(* CODESYS project CtaSysIO_2.0.0.0.library
   Description: Io System Library der CTA
   Version: 2.0.0.0
   Title: CtaSysIO
   Author: SIS
   DocFormat: reStructuredText
   LanguageModelAttribute: qualified-access-only
   Placeholder: CtaSysIO
   CompiledLibraryCompatibilityVersion: CODESYS V3.5 SP16 Patch 3
   Company: CTA
   DefaultNamespace: CtaSysIO

Project tree, tasks and I/O mapping:
  libraries: Standard, 3.5.18.0 (System); VisuDialogs, * (System); CtaSysConfig, 2.0.0.0 (CTA); CtaVisSymbols, 2.0.0.0 (CTA); VisuSymbols, 4.5.0.0 (System); CtaAppReport, 2.0.0.0 (CTA); CtaAppBmk, 2.0.0.0 (CTA); CtaVisHelp, 1.0.0.0 (CTA); CtaAppInfluxLog, 1.0.0.1 (CTA); SysCom, 3.5.17.0 (System); CtaAppBasic, 1.0.0.0 (CTA); Visu Utils, 4.5.0.0 (System)
  40 Visualizations/
    IO_FB/
      AI/
        visualisation SimAI_Temp
        visualisation SimAI
        visualisation SimAI_Temp_Querry
      AO/
        visualisation SimAO_Temp
        visualisation SimAO
        visualisation SimAO_Temp_Querry
      DI/
        visualisation SimDI
        visualisation SimDI_Temp
        visualisation SimDI_Temp_Querry
        SimValue/
          visualisation SimDI_Value
          visualisation SimDI_Value_Query
      DO/
        visualisation SimDO_Temp
        visualisation SimDO
        visualisation SimDO_Temp_Querry
        SimValue/
          visualisation SimDO_Value
          visualisation SimDO_Value_Query
      Simulation/
        visualisation Simulation
        visualisation ModulInfos
        visualisation SimulationInfos
        visualisation DIA_IO_CONFIG
      Parameter/
        visualisation VIS_IO_PARAMETER_BASE
        Parameter_AI/
          visualisation VIS_PARAMETER_AI
          visualisation VIS_PARAMETER_TEMP_AI
        Parameter_DI/
          visualisation VIS_PARAMETER_DI
          visualisation VIS_PARAMETER_TEMP_DI
        Parameter_AO/
          visualisation VIS_PARAMETER_AO
          visualisation VIS_PARAMETER_TEMP_AO
        Parameter_DO/
          visualisation VIS_PARAMETER_DO
          visualisation VIS_PARAMETER_TEMP_DO
      IO/
        visualisation SimIO
        visualisation SimIO_Query
        Invert/
          visualisation SimInvert
          visualisation SimInvert_Query
        visualisation SimIO_Temp
    IO_MANAGER/
      DEVICE/
        visualisation VIS_DEVICE
        visualisation VIS_DEVICE_QUERY
      visualisation DIA_IO_DEVICES
      NETZWERK/
        visualisation VIS_IO_DEVICES
        visualisation VIS_IO_DEVICES_NETWORK
    IO_TABLE/
      visualisation VIS_IO_TABLE
      visualisation VIS_IO_TABLE_QUERY
    IO_SLOT/
      visualisation VIS_IO_SLOT_IOS_ARRAY
      visualisation VIS_IO_SLOT_IOS_QUERY
      visualisation VIS_IO_SLOT_IOS
  30 Program Organization Units/
    IO_FB/
      IO/
        function block FB_IO [ST]: SELF, P_scfbIO_fbxSimulationLock, P_scfbIO_Simulation, ProSetInstancePathOnDynCreate, SELFPOINTER, IO_TYPE, IO_NR, PARENT, proSimVisu, proOK, proOkVisu, proPhysikalValueVisu, proIsSimLocked, proIsBOOL_IO, ADD_HAND, proLogName, DESTROY, BIG_SYBIL, LOW_SYBIL, SLOT_NR, REM_HAND
        function block FB_IO_TABLE [ST]: IO_NR, IO_TYPE, proSimVisu, SLOT_NR, proOkVisu, proPhysikalValueVisu
      AI/
        function block FB_AI [ST]: P_scfbAI_fbstPhysicalUnit, P_scfbAI_fbrMax, P_scfbAI_fbrMinPhysical, P_scfbAI_fbrMin, P_scfbAI_fbrPhysicalAlarm, P_scfbAI_fbrSimulationValue, P_scfbAI_fbrCorrectionValue, P_All_Init, proIsBOOL_IO, proPhysikalValueVisu, proPhysicalValue, proValue, metCyclicIoUpdate, metTrendLog, proAlUeberlauf, metConfig, proAlUnterlauf
      DO/
        function block FB_DO [ST]: P_scfbDO_fbxInvert, P_All_Init, P_scfbDO_fbxSimulationValue, metConfig, metTrendLog, proPhysikalValueVisu, proIsBOOL_IO, proValue, metCyclicIoUpdate
      AO/
        function block FB_AO [ST]: proIsBOOL_IO, P_All_Init, P_scfbAO_fbrMin, P_scfbAO_fbrMax, P_scfbAO_fbrSimulationValue, P_scfbAO_fbrMinPhysical, proValue, metCyclicIoUpdate, metTrendLog, metConfig, proPhysicalValue, proPhysikalValueVisu
      DI/
        function block FB_DI [ST]: metConfig, proPhysikalValueVisu, metCyclicIoUpdate, metTrendLog, P_scfbDI_fbxSimulationValue, P_scfbDI_fbxInvert, P_All_Init, proValue, proIsBOOL_IO
      FC/
        function fcScaleOut [ST]
        function fcScaleIn [ST]
    IO_DEVICE/
      function block FB_IO_DEVICE [ST]: AY_ITF_SLOT_VIS, BIG_SYBIL, LOW_SYBIL, ADDITION_DYN_SIZE, proVISU_DIA_NAME, IMAGE, COUNT, SELF, ADD_ERROR, ADD_SLOT, RELOAD_ARRAY, CHECK_IF_SLOT_EXIST, DEV_NR, DYN_SIZE, INSTANCE_PATH, ERROR, CREATE_SLOT, GET_SLOT, GET_IO, CHECK_ERROR, CHECK_HAND, ADD_HAND, HAND, REM_ERROR, REM_HAND, GET_STATE_READY_TO_SET_CONFIG, SET_STATE_READY_TO_SET_CONFIG, CHECK_SLOT, CONFIG_DONE, CHECK_SLOT_FAILS, SIM_IO_UPDATE, SIMULATION_ENABLED, FB_INIT, SIM_IO_TYPE
    IO_SLOT/
      function block FB_IO_SLOT [ST]: ADD_IO, CHECK_IF_IO_EXIST, CREATE_IO, GET_IO, BIG_SYBIL, LOW_SYBIL, PARENT, SELF, SLOT_NR, IMAGE, DYN_SIZE, RELOAD_ARRAY, AY_ITF_IO_VIS, SELFPOINTER, COUNT, ADD_ERROR, CHECK_SLOT
    IO_MANAGER/
      function block FB_IO_MANAGER [ST]: GET_DEVICE, GET_IO, AY_ITF_DEVICE_VIS, COUNT, ADD_DEVICE, CHECK_IF_DEVICE_EXIST, IMAGE, CHECK_SLOT
    FC/
      function FC_VIS_IO_TABLE [ST]
  00000000-0000-0000-0000-000000000000|D:\CoDeSys\LibrariesV3\trunk\Intern\CAA\CAA Template\3.4.0.0 draft\Placeholder.xml
  00000000-0000-0000-0000-000000000000|D:\CoDeSys\LibrariesV3\trunk\Intern\CAA\CAA Template\3.2.0.3 draft\Prefix.pdf
  00000000-0000-0000-0000-000000000000|D:\CoDeSys\LibrariesV3\trunk\Intern\CAA\CAA Template\3.5.2.0 draft\Placeholder.xml
  20 Structs/
    Parameter/
      data type scDI_Para
      data type scDO_Para
      data type scAI_Para
      data type scAO_Para
    data type enIOType
    data type enCheckIo
  50 Images/
  10 Documenation/
    global variables VersionHistory
    global variables readMe
  21 Interface/
    IO_MANAGER/
      interface ITF_IO_MANAGER: IMAGE, AY_ITF_DEVICE_VIS, COUNT
    IO_SLOT/
      interface ITF_IO_SLOT: BIG_SYBIL, LOW_SYBIL, SELF, PARENT, SLOT_NR, IMAGE, DYN_SIZE, GET_IO, CREATE_IO, AY_ITF_IO_VIS, RELOAD_ARRAY, SELFPOINTER, COUNT, CHECK_SLOT
    IO_DEVICE/
      interface ITF_IO_DEVICE: INSTANCE_PATH, ADD_ERROR, LOW_SYBIL, ERROR, ADD_HAND, SELF, HAND, IMAGE, DEV_NR, DYN_SIZE, RELOAD_ARRAY, COUNT, GET_IO, BIG_SYBIL, ADDITION_DYN_SIZE, proVISU_DIA_NAME, AY_ITF_SLOT_VIS, REM_ERROR, REM_HAND, GET_STATE_READY_TO_SET_CONFIG, SET_STATE_READY_TO_SET_CONFIG, CHECK_SLOT, SIM_IO_TYPE
    IO_FB/
      AI/
        interface ITF_AI: P_scfbAI_fbrPhysicalAlarm, P_scfbAI_fbrSimulationValue, P_scfbAI_fbstPhysicalUnit, P_scfbAI_fbrCorrectionValue, P_scfbAI_fbrMax, P_scfbAI_fbrMin, P_scfbAI_fbrMinPhysical, P_All_Init, proAlUeberlauf, proValue, proAlUnterlauf, metCyclicIoUpdate, proPhysicalValue
      AO/
        interface ITF_AO: proValue, proPhysicalValue, P_scfbAO_fbrMax, P_scfbAO_fbrMin, P_scfbAO_fbrMinPhysical, P_scfbAO_fbrSimulationValue, P_All_Init, metCyclicIoUpdate
      DI/
        interface ITF_DI: metCyclicIoUpdate, P_scfbDI_fbxInvert, P_scfbDI_fbxSimulationValue, P_All_Init, proValue
      DO/
        interface ITF_DO: proValue, metCyclicIoUpdate, P_scfbDO_fbxSimulationValue, P_All_Init, P_scfbDO_fbxInvert
      IO/
        interface ITF_IO: proIsBOOL_IO, P_scfbIO_Simulation, P_scfbIO_fbxSimulationLock, BIG_SYBIL, SELF, PARENT, IO_TYPE, proOK, ProSetInstancePathOnDynCreate, LOW_SYBIL, proOkVisu, IO_NR, SELFPOINTER, proPhysikalValueVisu, proSimVisu, proIsSimLocked, proLogName
        interface ITF_IO_TABLE: IO_TYPE, IO_NR, SLOT_NR, proOkVisu, proPhysikalValueVisu, proSimVisu
  11 Library Parameter/
    global variables Parameter
  12 Konstanten/
    global variables GlobalKonstant
  60 Textlisten/
    text list txtIOType
    text list txtWarning
    text list txtError
    text list txtPhysicalUnit
  13 Globale Variablen/
    global variables GVL_IO
  text list GlobalTextList
  5ce3da45-db07-42e7-a21c-a00fff4ed8f6|S:\_Temporär_SIS\CtaCodesysLibrary\01_Library\CtaSysIO\04_Image\0750_432.bmp
  5ce3da45-db07-42e7-a21c-a00fff4ed8f6|S:\_Temporär_SIS\CtaCodesysLibrary\01_Library\CtaSysIO\04_Image\0750_455.bmp
  5ce3da45-db07-42e7-a21c-a00fff4ed8f6|S:\_Temporär_SIS\CtaCodesysLibrary\01_Library\CtaSysIO\04_Image\0750_466.bmp
  5ce3da45-db07-42e7-a21c-a00fff4ed8f6|S:\_Temporär_SIS\CtaCodesysLibrary\01_Library\CtaSysIO\04_Image\0750_597.bmp
  5ce3da45-db07-42e7-a21c-a00fff4ed8f6|S:\_Temporär_SIS\CtaCodesysLibrary\01_Library\CtaSysIO\04_Image\0750_652.bmp
  5ce3da45-db07-42e7-a21c-a00fff4ed8f6|S:\_Temporär_SIS\CtaCodesysLibrary\01_Library\CtaSysIO\04_Image\0750_1415.bmp
  5ce3da45-db07-42e7-a21c-a00fff4ed8f6|S:\_Temporär_SIS\CtaCodesysLibrary\01_Library\CtaSysIO\04_Image\0750_8212.bmp
  5ce3da45-db07-42e7-a21c-a00fff4ed8f6|S:\_Temporär_SIS\CtaCodesysLibrary\01_Library\CtaSysIO\04_Image\0750_555.bmp
*)

// 20 Structs/Parameter/scDI_Para
TYPE scDI_Para :
	STRUCT
		xSimulationLock		:	BOOL;
		xInvert				:	BOOL;
	END_STRUCT
END_TYPE

// 20 Structs/Parameter/scDO_Para
TYPE scDO_Para :
	STRUCT
		xSimulationLock		:	BOOL;
		xInvert				:	BOOL;
	END_STRUCT
END_TYPE

// 20 Structs/Parameter/scAI_Para
TYPE scAI_Para :
	STRUCT
		xSimulationLock		:	BOOL;
		rMin				:	REAL;
		rMax				:	REAL;
		rMinPhysical		:	REAL;
		rPhysicalAlarm		:	REAL;
		rCorrectionValue	:	REAL;
		stPhysicalUnit		:	STRING(40);
	END_STRUCT
END_TYPE

// 20 Structs/Parameter/scAO_Para
TYPE scAO_Para :
	STRUCT
		xSimulationLock		:	BOOL;
		rMin				:	REAL;
		rMax				:	REAL;
		rMinPhysical		:	REAL;
	END_STRUCT
END_TYPE

// 20 Structs/enIOType
{attribute 'qualified_only'}
{attribute 'to_string'}

TYPE enIOType :
(
	Unknown 		:= 0,
	Digital_IN		:= 1,
	Digital_OUT		:= 2,	
	DC_0_10V_OUT	:= 3,
	DC_4_20mA_OUT	:= 4,
	DC_0_10V_IN		:= 5,
	DC_4_20mA_IN	:= 6,
	OHM				:= 7,
	DC_0_20mA_OUT	:= 8,
	TEMPERATUR		:= 9,
	DC_0_20mA_IN	:= 10
);
END_TYPE

// 20 Structs/enCheckIo
TYPE enCheckIo :
(
		DI_IO	:=	0,
		AI_IO	:=	1,
		DO_IO	:=	2,
		AO_IO	:=	3
);
END_TYPE

// 10 Documenation/VersionHistory
(* 

.. image:: ../../Images/CTA_Logo.jpg
   :align: right
   :width: 15% 

**Vorlage**   


============ =========== =========== ============================================
**Date**     **Version** **Author**  **Change**
------------ ----------- ----------- --------------------------------------------
04.03.2021   0.0.0.0     SIS         Vorlage erstellt

============ =========== =========== ============================================


*)
VAR_GLOBAL
    stInfo : STRING:= '0.0.0.0, Vorlage, CTA';
END_VAR

// 10 Documenation/readMe
(*

**ReadMe**
 
|	**Empfehlung**
|
|	Dokumentrieren Sie die Library für eine nachhaltige Entwicklung
|     
| *Beispiel*
| 
| Dies ist die Vorlage Library der CTA. Erstellen Sie ihre Library anhand dieser Vorlage.
*)

VAR_GLOBAL
    xReadMeDone              :   BOOL;
END_VAR

// 13 Globale Variablen/GVL_IO
{attribute 'qualified_only'}
VAR_GLOBAL	
	FB_IO_MANAGER : FB_IO_MANAGER;
END_VAR

// 11 Library Parameter/Parameter
{attribute 'qualified_only'}
VAR_GLOBAL CONSTANT
	SPS_BMK_ID        		: STRING(20)   := 'SPS';
	MAX_NUM_OF_DI			: INT := 200;
	MAX_NUM_OF_DO			: INT := 200;
	MAX_NUM_OF_AI			: INT := 100;
	MAX_NUM_OF_AO			: INT := 100;	
	                		
	MAX_NUM_OF_IOS			: INT := MAX_NUM_OF_DI + MAX_NUM_OF_DO + MAX_NUM_OF_AI + MAX_NUM_OF_AO;
	
	MAX_NUM_OF_COMTYPES		: INT := 10;
END_VAR

// 12 Konstanten/GlobalKonstant
{attribute 'qualified_only'}
VAR_GLOBAL CONSTANT
    stWarningTextList   :   STRING  := 'CtaSysIO.txtWarning';
    stErrorTextList     :   STRING  := 'CtaSysIO.txtError';
END_VAR

// 30 Program Organization Units/IO_DEVICE/FB_IO_DEVICE
{attribute 'reflection'}
FUNCTION_BLOCK FB_IO_DEVICE EXTENDS CtaAppBmk.fbBMK IMPLEMENTS ITF_IO_DEVICE
VAR_INPUT
	usiDevNr	:	USINT;
END_VAR
VAR_OUTPUT
	xReadyToIoConfig			:	BOOL;
	xConfigDone					:	BOOL;
	xError						:	BOOL;
	xSlotMissmatch				:	BOOL;
	xHand						:	BOOL;
	udiDynMem					:	UDINT;	
END_VAR
VAR
	_IMAGE						:	STRING;
	
	_ITF_BIG_SYBIL				:	ITF_IO_DEVICE;
	_ITF_LOW_SYBIL				:	ITF_IO_DEVICE;
	                			
	_BASE_SLOT					:	ITF_IO_SLOT;
	_TEMP_REG_SLOT				:	ITF_IO_SLOT;
	_NEXT_SLOT_LAST_GET			:	ITF_IO_SLOT;	
	
	_COUNT						:	UINT;
	_udiDynMemTemp				:	UDINT;	
	_ayITF_SLOTS				:	ARRAY[0..255] OF ITF_IO_SLOT;
	_ayITF_SLOT_VIS				:	ARRAY[1..10] OF ITF_IO_SLOT;
	
	_ALLOW_SIMULATION			:	BOOL;
	_ENABLE_SIMULATION			:	BOOL;
	_INIT_DONE_SIMULATION		:	BOOL;
	
	udiCountError				:	UDINT;	
	udiCountHand				:	UDINT;
	udiCountCheckSlotFails		:	UDINT;
	udiCountCheckSlotFailsOld	:	UDINT;
	
END_VAR

xSlotMissmatch 	:= CHECK_SLOT_FAILS();
xHand 			:= CHECK_HAND();
xError 			:= CHECK_ERROR();

SIM_IO_UPDATE();

PROPERTY AY_ITF_SLOT_VIS : ARRAY[1..10] OF ITF_IO_SLOT;
GET
AY_ITF_SLOT_VIS := _ayITF_SLOT_VIS;
END_GET
END_PROPERTY

{attribute 'estimated-stack-usage' := '104'}
PROPERTY BIG_SYBIL : ITF_IO_DEVICE
SET
_ITF_BIG_SYBIL := BIG_SYBIL;
IF __QUERYINTERFACE(_ITF_BIG_SYBIL,_ITF_BIG_SYBIL) THEN
	IF _ITF_BIG_SYBIL.LOW_SYBIL <> SELF THEN
		_ITF_BIG_SYBIL.LOW_SYBIL := THIS^;
	END_IF;
END_IF;
END_SET
GET
BIG_SYBIL := _ITF_BIG_SYBIL;
END_GET
END_PROPERTY

{attribute 'estimated-stack-usage' := '104'}
PROPERTY LOW_SYBIL : ITF_IO_DEVICE
GET
LOW_SYBIL := _ITF_LOW_SYBIL;
END_GET
SET
_ITF_LOW_SYBIL := LOW_SYBIL;
IF __QUERYINTERFACE(_ITF_LOW_SYBIL,_ITF_LOW_SYBIL) THEN
	IF _ITF_LOW_SYBIL.BIG_SYBIL <> SELF THEN
		_ITF_LOW_SYBIL.BIG_SYBIL := THIS^;
	END_IF;
END_IF;
END_SET
END_PROPERTY

PROPERTY ADDITION_DYN_SIZE : DINT
SET
VAR
	diTemp	:	DINT;
END_VAR
IF ADDITION_DYN_SIZE > 0 THEN
	_udiDynMemTemp := _udiDynMemTemp + TO_UDINT(ADDITION_DYN_SIZE);
ELSE
	_udiDynMemTemp := _udiDynMemTemp - TO_UDINT(ADDITION_DYN_SIZE);
END_IF;
udiDynMem	:= MAX(udiDynMem,_udiDynMemTemp);
END_SET
END_PROPERTY

PROPERTY proVISU_DIA_NAME : STRING
GET
proVISU_DIA_NAME := '';
END_GET
END_PROPERTY

PROPERTY IMAGE : STRING
GET
IMAGE := _IMAGE;
END_GET
SET
_IMAGE := IMAGE;
END_SET
END_PROPERTY

PROPERTY COUNT : UINT
GET
COUNT := _COUNT;
END_GET
END_PROPERTY

PROPERTY SELF : ITF_IO_DEVICE
GET
SELF := THIS^;
END_GET
END_PROPERTY

METHOD ADD_ERROR
VAR_INPUT
END_VAR
udiCountError := udiCountError + 1;
END_METHOD

METHOD ADD_SLOT
VAR_INPUT
	ITF_SLOT_IN		:	ITF_IO_SLOT;
END_VAR
VAR
	ITF_TEMP		:	ITF_IO_SLOT;
	ITF_TEMP_BIG	:	ITF_IO_SLOT;
	ITF_TEMP_LOW	:	ITF_IO_SLOT;
	xDone			:	BOOL;
END_VAR
(* Check if Valid Interface Input *)
IF __QUERYINTERFACE(ITF_SLOT_IN,ITF_SLOT_IN) THEN
	ITF_SLOT_IN.PARENT := THIS^;
	IF TO_DINT(ITF_SLOT_IN.SLOT_NR) >= LOWER_BOUND(_ayITF_SLOTS,1) AND
	   TO_DINT(ITF_SLOT_IN.SLOT_NR) <= UPPER_BOUND(_ayITF_SLOTS,1) THEN
	   _ayITF_SLOTS[ITF_SLOT_IN.SLOT_NR] := ITF_SLOT_IN;
	END_IF;
	(* Check if Valid Interface Base*)
	IF __QUERYINTERFACE(_BASE_SLOT,_BASE_SLOT) THEN
		(* Check if Valid Interface Temporary registration *)
		IF __QUERYINTERFACE(_TEMP_REG_SLOT,ITF_TEMP) THEN
			REPEAT
				(* Get Big Sybil of registration *)
				IF __QUERYINTERFACE(ITF_TEMP.BIG_SYBIL,ITF_TEMP_BIG) THEN
					(* Check if Adress is Lower *)
					IF ITF_SLOT_IN.SLOT_NR <= ITF_TEMP.SLOT_NR THEN
						(* Check if Adress is Bigger and update if yes*)
						IF ITF_SLOT_IN.SLOT_NR >= ITF_TEMP_BIG.SLOT_NR THEN
							ITF_SLOT_IN.BIG_SYBIL := ITF_TEMP.BIG_SYBIL;
							ITF_SLOT_IN.LOW_SYBIL := ITF_TEMP;
							xDone	 := TRUE;							
						END_IF;
					(* Adress is Bigger update *)
					ELSE
						IF __QUERYINTERFACE(ITF_TEMP.LOW_SYBIL,ITF_TEMP_LOW) THEN
							IF 	ITF_SLOT_IN.SLOT_NR <= ITF_TEMP_LOW.SLOT_NR THEN
								ITF_SLOT_IN.LOW_SYBIL := ITF_TEMP.LOW_SYBIL;
								ITF_SLOT_IN.BIG_SYBIL := ITF_TEMP;
								xDone	 := TRUE;
							END_IF;
						ELSE
							ITF_SLOT_IN.LOW_SYBIL := ITF_TEMP.LOW_SYBIL;
							ITF_SLOT_IN.BIG_SYBIL := ITF_TEMP;
							xDone	 := TRUE;
							(* Update Registation Job if temp is the last one *)
							IF ITF_TEMP = _TEMP_REG_SLOT THEN
								_TEMP_REG_SLOT := ITF_SLOT_IN;
								_TEMP_REG_SLOT.LOW_SYBIL := 0;
							END_IF;
						END_IF;
					END_IF;
				(* Interface is same as the Base*)
				ELSIF ITF_TEMP = _BASE_SLOT THEN
					(* Check if the Input Interface needs to be the new base*)
					IF ITF_SLOT_IN.SLOT_NR <= ITF_TEMP.SLOT_NR THEN 
						ITF_SLOT_IN.LOW_SYBIL := ITF_TEMP;
						_BASE_SLOT 				:= ITF_SLOT_IN;
						_BASE_SLOT.BIG_SYBIL 	:= 0;
						xDone	 				:= TRUE; 
					ELSE
						(* Update Registation Job if temp is the last one *)
						IF ITF_TEMP = _TEMP_REG_SLOT THEN
							_TEMP_REG_SLOT				:= ITF_SLOT_IN;
							_TEMP_REG_SLOT.LOW_SYBIL 	:= 0;
						END_IF
						ITF_SLOT_IN.LOW_SYBIL := _BASE_SLOT.LOW_SYBIL;
						_BASE_SLOT.LOW_SYBIL 	:= ITF_SLOT_IN;
					END_IF;
				END_IF;
				(* Get Next Interface to Check*)
				__QUERYINTERFACE(ITF_TEMP.BIG_SYBIL,ITF_TEMP);
			UNTIL xDone OR ITF_TEMP = 0 
			END_REPEAT
		ELSE
			(* Set Base Low sybill on second call*)
			_BASE_SLOT.LOW_SYBIL 	:= ITF_SLOT_IN;
			_TEMP_REG_SLOT			:= ITF_SLOT_IN;		
		END_IF;		
	ELSE
		(* Set Base on first call*)
		_BASE_SLOT 		:= ITF_SLOT_IN;
		_TEMP_REG_SLOT 	:= ITF_SLOT_IN;
	END_IF;
	(* Count Jobs *)
	_COUNT := _COUNT + 1;
	THIS^.RELOAD_ARRAY(TRUE,FALSE,FALSE);
END_IF;
END_METHOD

METHOD RELOAD_ARRAY
VAR_INPUT
	xInit	: BOOL;
	xLoadNext10	: BOOL;
	xLoadLast10	: BOOL;
END_VAR
VAR
	diFor				:	DINT;
	ITF_TEMP_CLIENT_VIS	:	ITF_IO_SLOT;
	ITF_TEMP_SAFE		:	ITF_IO_SLOT;
	ITF_TEMP_LAST_VALID	:	ITF_IO_SLOT;
END_VAR
(* Init Array *)
IF xInit THEN
	_ayITF_SLOT_VIS[LOWER_BOUND(_ayITF_SLOT_VIS,1)] := _BASE_SLOT;
	FOR diFor := LOWER_BOUND(_ayITF_SLOT_VIS,1) TO UPPER_BOUND(_ayITF_SLOT_VIS,1) -1 DO
		IF __QUERYINTERFACE(_ayITF_SLOT_VIS[diFor],ITF_TEMP_CLIENT_VIS) THEN
			_ayITF_SLOT_VIS[diFor + 1]	:= _ayITF_SLOT_VIS[diFor].LOW_SYBIL;
		ELSE
			_ayITF_SLOT_VIS[diFor + 1] := 0;
		END_IF;	
	END_FOR;
(* Load Next 10 *)
ELSIF xLoadNext10 THEN
	IF __QUERYINTERFACE(_ayITF_SLOT_VIS[UPPER_BOUND(_ayITF_SLOT_VIS,1)],ITF_TEMP_CLIENT_VIS) THEN
		_ayITF_SLOT_VIS[LOWER_BOUND(_ayITF_SLOT_VIS,1)] := ITF_TEMP_CLIENT_VIS.LOW_SYBIL;
		FOR diFor := LOWER_BOUND(_ayITF_SLOT_VIS,1) TO UPPER_BOUND(_ayITF_SLOT_VIS,1) -1 DO
			IF __QUERYINTERFACE(_ayITF_SLOT_VIS[diFor],ITF_TEMP_CLIENT_VIS) THEN
				_ayITF_SLOT_VIS[diFor + 1]	:= _ayITF_SLOT_VIS[diFor].LOW_SYBIL;
			ELSE
				_ayITF_SLOT_VIS[diFor + 1] := 0;
			END_IF;	
		END_FOR;
	END_IF;
(* Load Last 10 *)
ELSIF xLoadLast10 THEN
	IF __QUERYINTERFACE(_ayITF_SLOT_VIS[LOWER_BOUND(_ayITF_SLOT_VIS,1)],ITF_TEMP_CLIENT_VIS) THEN
		IF __QUERYINTERFACE(_ayITF_SLOT_VIS[LOWER_BOUND(_ayITF_SLOT_VIS,1)].BIG_SYBIL,ITF_TEMP_SAFE) THEN
			_ayITF_SLOT_VIS[UPPER_BOUND(_ayITF_SLOT_VIS,1)] := ITF_TEMP_CLIENT_VIS.BIG_SYBIL;
			FOR diFor := UPPER_BOUND(_ayITF_SLOT_VIS,1) TO LOWER_BOUND(_ayITF_SLOT_VIS,1) + 1 BY -1 DO 
				IF __QUERYINTERFACE(_ayITF_SLOT_VIS[diFor],ITF_TEMP_CLIENT_VIS) THEN
					ITF_TEMP_LAST_VALID  			:= _ayITF_SLOT_VIS[diFor];
					_ayITF_SLOT_VIS[diFor - 1]	:= _ayITF_SLOT_VIS[diFor].BIG_SYBIL;
				ELSE
					(* Resort if new ones Inside *)
					_ayITF_SLOT_VIS[LOWER_BOUND(_ayITF_SLOT_VIS,1)] := ITF_TEMP_LAST_VALID;
					FOR diFor := LOWER_BOUND(_ayITF_SLOT_VIS,1) TO UPPER_BOUND(_ayITF_SLOT_VIS,1) -1 DO
						IF __QUERYINTERFACE(_ayITF_SLOT_VIS[diFor],ITF_TEMP_CLIENT_VIS) THEN
							_ayITF_SLOT_VIS[diFor + 1]	:= _ayITF_SLOT_VIS[diFor].LOW_SYBIL;
						ELSE
							_ayITF_SLOT_VIS[diFor + 1] := 0;
						END_IF;	
					END_FOR;					
				END_IF;	
			END_FOR;
		END_IF;
	END_IF;	
END_IF;
END_METHOD

METHOD CHECK_IF_SLOT_EXIST : BOOL
VAR_INPUT
	_usiSlotNr			: 	USINT;
END_VAR
VAR
	_TEMP_CHK_SLOT	:	ITF_IO_SLOT;
	udiSafe			:	UDINT;
END_VAR
IF __QUERYINTERFACE(_BASE_SLOT,_TEMP_CHK_SLOT) THEN
	REPEAT 
		IF _TEMP_CHK_SLOT.SLOT_NR = _usiSlotNr THEN
			CHECK_IF_SLOT_EXIST := TRUE;
		END_IF;
		_TEMP_CHK_SLOT := _TEMP_CHK_SLOT.LOW_SYBIL;
		udiSafe	:= udiSafe + 1;
	UNTIL CHECK_IF_SLOT_EXIST OR _TEMP_CHK_SLOT = 0 OR udiSafe >= 16#FFFFFFFE
	END_REPEAT
ELSE
	CHECK_IF_SLOT_EXIST := FALSE;
END_IF
END_METHOD

PROPERTY DEV_NR : USINT
GET
DEV_NR := usiDevNr;
END_GET
END_PROPERTY

PROPERTY DYN_SIZE : UDINT
GET
DYN_SIZE := udiDynMem;
END_GET
END_PROPERTY

PROPERTY INSTANCE_PATH : STRING(255)
GET
INSTANCE_PATH := stInstancePath;
END_GET
END_PROPERTY

PROPERTY ERROR : BOOL
GET
ERROR := xError;
END_GET
END_PROPERTY

METHOD CREATE_SLOT : BOOL
VAR_INPUT
	_usiSlotNr			: 	USINT;
	_stSlotImage		:	STRING;
END_VAR
VAR	
	pFbIO				:	POINTER TO FB_IO_SLOT;
END_VAR
IF NOT CHECK_IF_SLOT_EXIST(_usiSlotNr) THEN
	pFbIO := __NEW(FB_IO_SLOT);
	IF pFbIO <> 0 THEN
		_udiDynMemTemp 							:= _udiDynMemTemp + SIZEOF(FB_IO);
		udiDynMem								:= MAX(udiDynMem,_udiDynMemTemp);
		pFbIO^.SLOT_NR		 					:= _usiSlotNr;
		pFbIO^.IMAGE		 					:= _stSlotImage;
		ADD_SLOT(pFbIO^);
	ELSE
		ADD_ERROR();
	END_IF;
END_IF;
END_METHOD

METHOD GET_SLOT : ITF_IO_SLOT
VAR_INPUT
	_usiSlotNr			: 	USINT;
END_VAR
VAR
	_TEMP_GET_SLOT	:	ITF_IO_SLOT;
	udiSafe			:	UDINT;
	xNextIoInUse	:	BOOL;
END_VAR
IF TO_DINT(_usiSlotNr) >= LOWER_BOUND(_ayITF_SLOTS,1) AND
   TO_DINT(_usiSlotNr) <= UPPER_BOUND(_ayITF_SLOTS,1) THEN
   GET_SLOT := _ayITF_SLOTS[_usiSlotNr];
END_IF;

IF GET_SLOT = 0 THEN
	IF __QUERYINTERFACE(_NEXT_SLOT_LAST_GET,_TEMP_GET_SLOT) THEN
		xNextIoInUse := TRUE;
	ELSIF __QUERYINTERFACE(_BASE_SLOT,_TEMP_GET_SLOT) THEN
		xNextIoInUse := FALSE;
	END_IF;
	
	IF __QUERYINTERFACE(_TEMP_GET_SLOT,_TEMP_GET_SLOT) THEN
		REPEAT 
			IF _TEMP_GET_SLOT.SLOT_NR = _usiSlotNr THEN
				GET_SLOT := _TEMP_GET_SLOT;
			END_IF;
			_TEMP_GET_SLOT	 	:= _TEMP_GET_SLOT.LOW_SYBIL;
			_NEXT_SLOT_LAST_GET	:= _TEMP_GET_SLOT;
			IF _TEMP_GET_SLOT = 0 AND xNextIoInUse THEN
				__QUERYINTERFACE(_BASE_SLOT,_TEMP_GET_SLOT);
				xNextIoInUse := FALSE;
			END_IF;
			udiSafe	:= udiSafe + 1;
		UNTIL GET_SLOT <> 0 OR _TEMP_GET_SLOT = 0 OR udiSafe >= 16#FFFFFFFE
		END_REPEAT
	ELSE
		GET_SLOT := 0;
	END_IF;
END_IF;
END_METHOD

METHOD GET_IO : ITF_IO
VAR_INPUT
	_usiSlotNr			: 	USINT;
	_usiIoNr			: 	USINT;
END_VAR	
VAR
	_TEMP_GET_SLOT	:	ITF_IO_SLOT;
	_TEMP_GET_IO		:	ITF_IO;
	udiSafe				:	UDINT;
END_VAR
IF __QUERYINTERFACE(GET_SLOT(_usiSlotNr),_TEMP_GET_SLOT) THEN
	GET_IO := _TEMP_GET_SLOT.GET_IO(_usiIoNr);
END_IF;
END_METHOD

METHOD CHECK_ERROR : BOOL
VAR_INPUT
END_VAR
CHECK_ERROR := udiCountError <> 0;
END_METHOD

METHOD CHECK_HAND : BOOL
VAR_INPUT
END_VAR
CHECK_HAND := udiCountHand <> 0;
END_METHOD

METHOD ADD_HAND
VAR_INPUT
END_VAR
udiCountHand := udiCountHand + 1;
END_METHOD

PROPERTY HAND : BOOL
GET
HAND := xHand;
END_GET
END_PROPERTY

METHOD REM_ERROR
VAR_INPUT
END_VAR
VAR
	ITF_IO_DEVICE_TEMP	:	ITF_IO_DEVICE;
END_VAR
udiCountError := udiCountError - 1;
END_METHOD

METHOD REM_HAND
VAR_INPUT
END_VAR
VAR
	ITF_IO_DEVICE_TEMP	:	ITF_IO_DEVICE;
END_VAR
udiCountHand := udiCountHand - 1;
END_METHOD

PROPERTY GET_STATE_READY_TO_SET_CONFIG : BOOL
GET
GET_STATE_READY_TO_SET_CONFIG := xReadyToIoConfig;
END_GET
END_PROPERTY

PROPERTY SET_STATE_READY_TO_SET_CONFIG : BOOL
SET
xReadyToIoConfig := SET_STATE_READY_TO_SET_CONFIG;
END_SET
END_PROPERTY

METHOD CHECK_SLOT : BOOL
VAR_INPUT
	_usiSlotNr		: 	USINT;
	enCheckIoIn		:	enCheckIo;
	usiAnzIoType	:	USINT;
END_VAR
VAR
	ITF_SLOT		: 	ITF_IO_SLOT;
END_VAR
ITF_SLOT := GET_SLOT(_usiSlotNr);
IF __QUERYINTERFACE(ITF_SLOT,ITF_SLOT) THEN
	CHECK_SLOT := ITF_SLOT.CHECK_SLOT(enCheckIoIn,usiAnzIoType);
ELSE
	CHECK_SLOT := FALSE;
END_IF;
IF NOT CHECK_SLOT AND xConfigDone THEN
	udiCountCheckSlotFails := udiCountCheckSlotFails + 1;
END_IF;
END_METHOD

PROPERTY CONFIG_DONE : BOOL
SET
xConfigDone := CONFIG_DONE;
END_SET
GET
CONFIG_DONE := xConfigDone;
END_GET
END_PROPERTY

METHOD INTERNAL CHECK_SLOT_FAILS : BOOL
VAR_INPUT
END_VAR
IF udiCountCheckSlotFails > 0 AND udiCountCheckSlotFails <> udiCountCheckSlotFailsOld THEN
	ADD_ERROR();
	udiCountCheckSlotFailsOld := udiCountCheckSlotFails;
ELSIF udiCountCheckSlotFails = 0 AND udiCountCheckSlotFails <> udiCountCheckSlotFailsOld THEN
	udiCountCheckSlotFailsOld := udiCountCheckSlotFails;
	REM_ERROR();
END_IF;
CHECK_SLOT_FAILS := udiCountCheckSlotFails > 0;
udiCountCheckSlotFails := 0;
END_METHOD

METHOD SIM_IO_UPDATE
VAR
	_ITF_SLOT_SIM	:	ITF_IO_SLOT;
	_ITF_IO_SIM		:	ITF_IO;
	_ITF_IO_SIM_DI	:	ITF_DI;
	_ITF_IO_SIM_AI	:	ITF_AI;
	_ITF_IO_SIM_DO	:	ITF_DO;
	_ITF_IO_SIM_AO	:	ITF_AO;
END_VAR
VAR
	usiFor			:	USINT;
END_VAR
// Prüfen, ob die Simulation aktiviert ist und die Initialisierung abgeschlossen wurde
IF SIMULATION_ENABLED AND CONFIG_DONE THEN

	// Prüfen, ob das Basismodul (_BASE_SLOT) das Interface für simulierte Slots (_ITF_SLOT_SIM) unterstützt
	IF __QUERYINTERFACE(_BASE_SLOT, _ITF_SLOT_SIM) THEN

		// Wiederhole, solange es noch simulierte Slots gibt
		REPEAT
			// Iteriere über alle IOs im aktuellen simulierten Slot
			FOR usiFor := 1 TO _ITF_SLOT_SIM.COUNT DO
				// Hole das IO-Element an der aktuellen Position
				_ITF_IO_SIM := _ITF_SLOT_SIM.GET_IO(usiFor);

				// Prüfen, ob es sich um ein digitales Eingangsmodul handelt
				IF __QUERYINTERFACE(_ITF_IO_SIM, _ITF_IO_SIM_DI) THEN
					// Zyklisches Update für digitales Eingangssignal ausführen
					_ITF_IO_SIM_DI.metCyclicIoUpdate(FALSE, TRUE);

				// Prüfen, ob es sich um ein analoges Eingangsmodul handelt
				ELSIF __QUERYINTERFACE(_ITF_IO_SIM, _ITF_IO_SIM_AI) THEN
					// Zyklisches Update für analoges Eingangssignal ausführen
					_ITF_IO_SIM_AI.metCyclicIoUpdate(TRUE, 0, FALSE, FALSE);

				// Prüfen, ob es sich um ein digitales Ausgangsmodul handelt
				ELSIF __QUERYINTERFACE(_ITF_IO_SIM, _ITF_IO_SIM_DO) THEN
					// Zyklisches Update für digitales Ausgangssignal ausführen
					_ITF_IO_SIM_DO.metCyclicIoUpdate(TRUE);

				// Prüfen, ob es sich um ein analoges Ausgangsmodul handelt
				ELSIF __QUERYINTERFACE(_ITF_IO_SIM, _ITF_IO_SIM_AO) THEN
					// Zyklisches Update für analoges Ausgangssignal ausführen
					_ITF_IO_SIM_AO.metCyclicIoUpdate(TRUE);
				END_IF;
			END_FOR;

			// Zum nächsten simulierten Slot wechseln (Linked-List-Mechanismus oder ähnliche Struktur)
			_ITF_SLOT_SIM := _ITF_SLOT_SIM.LOW_SYBIL;

		// Wiederhole solange, bis kein weiterer Slot vorhanden ist (d.h. Ende der Kette erreicht)
		UNTIL _ITF_SLOT_SIM = 0
		END_REPEAT;
	END_IF;
END_IF;;
END_METHOD

(* Enable Simulation *)
PROPERTY SIMULATION_ENABLED : BOOL
GET
SIMULATION_ENABLED := _ENABLE_SIMULATION;
END_GET
END_PROPERTY

//FB_Init ist immer implizit verfügbar und wird primär für die Initialisierung verwendet.
//Der Rückgabewert wird nicht ausgewertet. Für gezielte Einflussnahme können Sie
//die Methoden explizit deklarieren und darin mit dem Standard-Initialisierungscode 
//zusätzlichen Code bereitstellen. Sie können den Rückgabewert auswerten.
METHOD FB_Init: BOOL
VAR_INPUT    
	bInitRetains				: BOOL; // TRUE: Die Retain-Variablen werden initialisiert (Reset warm / Reset kalt)    
	bInCopyCode					: BOOL;  // TRUE: Die Instanz wird danach in den Kopiercode kopiert (Online-Change)
	xEnableSimulationOnReboot	: BOOL;
END_VAR
_ENABLE_SIMULATION := xEnableSimulationOnReboot;
END_METHOD

METHOD SIM_IO_TYPE
VAR_INPUT
	_usiSlotNr		: 	USINT;
	enSimIoTypeIn	:	enIOType;
	usiAnzIoType	:	USINT;
	_stSlotImage	:	STRING;
END_VAR
VAR
	usiFor			:	USINT;
	ITF_SLOT_TEMP	:	ITF_IO_SLOT;
END_VAR
IF SIMULATION_ENABLED THEN
	IF _usiSlotNr > _COUNT THEN
		CREATE_SLOT(_usiSlotNr,_stSlotImage);
		FOR usiFor := 1 TO usiAnzIoType DO
			ITF_SLOT_TEMP := GET_SLOT(_usiSlotNr);
			IF __QUERYINTERFACE(ITF_SLOT_TEMP,ITF_SLOT_TEMP) THEN
				ITF_SLOT_TEMP.CREATE_IO(usiFor,enSimIoTypeIn);
			END_IF;
		END_FOR;
	ELSE
		_INIT_DONE_SIMULATION := TRUE;
	END_IF;
END_IF;
END_METHOD

END_FUNCTION_BLOCK

// 21 Interface/IO_DEVICE/ITF_IO_DEVICE
INTERFACE ITF_IO_DEVICE EXTENDS CtaAppBmk.ITF_BMK

PROPERTY INSTANCE_PATH : STRING(255)
GET
END_GET
END_PROPERTY

METHOD ADD_ERROR
VAR_INPUT
END_VAR
END_METHOD

{attribute 'estimated-stack-usage' := '104'}
PROPERTY LOW_SYBIL : ITF_IO_DEVICE
SET
END_SET
GET
END_GET
END_PROPERTY

PROPERTY ERROR : BOOL
GET
END_GET
END_PROPERTY

METHOD ADD_HAND
VAR_INPUT
END_VAR
END_METHOD

PROPERTY SELF : ITF_IO_DEVICE
GET
END_GET
END_PROPERTY

PROPERTY HAND : BOOL
GET
END_GET
END_PROPERTY

PROPERTY IMAGE : STRING
GET
END_GET
END_PROPERTY

PROPERTY DEV_NR : USINT
GET
END_GET
END_PROPERTY

PROPERTY DYN_SIZE : UDINT
GET
END_GET
END_PROPERTY

METHOD RELOAD_ARRAY
VAR_INPUT
	xInit	: BOOL;
	xLoadNext10	: BOOL;
	xLoadLast10	: BOOL;
END_VAR
END_METHOD

PROPERTY COUNT : UINT
GET
END_GET
END_PROPERTY

METHOD GET_IO : ITF_IO
VAR_INPUT
	_usiSlotNr			: 	USINT;
	_usiIoNr			: 	USINT;
END_VAR
END_METHOD

{attribute 'estimated-stack-usage' := '104'}
PROPERTY BIG_SYBIL : ITF_IO_DEVICE
GET
END_GET
SET
END_SET
END_PROPERTY

PROPERTY ADDITION_DYN_SIZE : DINT
SET
END_SET
END_PROPERTY

PROPERTY proVISU_DIA_NAME : STRING
GET
END_GET
END_PROPERTY

PROPERTY AY_ITF_SLOT_VIS : ARRAY[1..10] OF ITF_IO_SLOT;
GET
END_GET
END_PROPERTY

METHOD REM_ERROR
VAR_INPUT
END_VAR
END_METHOD

METHOD REM_HAND
VAR_INPUT
END_VAR
END_METHOD

PROPERTY GET_STATE_READY_TO_SET_CONFIG : BOOL
GET
END_GET
END_PROPERTY

PROPERTY INTERNAL SET_STATE_READY_TO_SET_CONFIG : BOOL
SET
END_SET
END_PROPERTY

METHOD CHECK_SLOT : BOOL
VAR_INPUT
	_usiSlotNr		: 	USINT;
	enCheckIoIn		:	enCheckIo;
	usiAnzIoType	:	USINT;
END_VAR
END_METHOD

METHOD SIM_IO_TYPE
VAR_INPUT
	_usiSlotNr		: 	USINT;
	enSimIoTypeIn	:	enIOType;
	usiAnzIoType	:	USINT;
	_stSlotImage	:	STRING;
END_VAR
END_METHOD

END_INTERFACE

// 21 Interface/IO_FB/IO/ITF_IO
INTERFACE ITF_IO EXTENDS ITF_IO_TABLE

PROPERTY proIsBOOL_IO : BOOL
GET
END_GET
END_PROPERTY

PROPERTY P_scfbIO_Simulation : CtaSysConfig.ITF_DATATYPE
GET
END_GET
END_PROPERTY

PROPERTY P_scfbIO_fbxSimulationLock : CtaSysConfig.ITF_DATATYPE
GET
END_GET
END_PROPERTY

PROPERTY BIG_SYBIL : ITF_IO
SET
END_SET
GET
END_GET
END_PROPERTY

PROPERTY SELF : ITF_IO
GET
END_GET
END_PROPERTY

PROPERTY PARENT : ITF_IO_SLOT
SET
END_SET
GET
END_GET
END_PROPERTY

PROPERTY IO_TYPE : enIOType
GET
END_GET
SET
END_SET
END_PROPERTY

PROPERTY proOK : BOOL
GET
END_GET
END_PROPERTY

PROPERTY ProSetInstancePathOnDynCreate : STRING(255);
SET
END_SET
END_PROPERTY

PROPERTY LOW_SYBIL : ITF_IO
SET
END_SET
GET
END_GET
END_PROPERTY

PROPERTY proOkVisu : STRING
GET
END_GET
END_PROPERTY

PROPERTY IO_NR : USINT
SET
END_SET
GET
END_GET
END_PROPERTY

{attribute 'monitoring' := 'call'}
PROPERTY SELFPOINTER : POINTER TO FB_IO
GET
END_GET
END_PROPERTY

PROPERTY proPhysikalValueVisu : STRING(6)
GET
END_GET
SET
END_SET
END_PROPERTY

PROPERTY proSimVisu : STRING
GET
END_GET
END_PROPERTY

PROPERTY proIsSimLocked : BOOL
GET
END_GET
END_PROPERTY

PROPERTY proLogName : STRING(100)
GET
END_GET
END_PROPERTY

END_INTERFACE

// 21 Interface/IO_FB/IO/ITF_IO_TABLE
INTERFACE ITF_IO_TABLE EXTENDS __System.IQueryinterface

PROPERTY IO_TYPE : enIOType
GET
END_GET
SET
END_SET
END_PROPERTY

PROPERTY IO_NR : USINT
SET
END_SET
GET
END_GET
END_PROPERTY

PROPERTY SLOT_NR : USINT
SET
END_SET
GET
END_GET
END_PROPERTY

PROPERTY proOkVisu : STRING
GET
END_GET
END_PROPERTY

PROPERTY proPhysikalValueVisu : STRING(6)
GET
END_GET
SET
END_SET
END_PROPERTY

PROPERTY proSimVisu : STRING
GET
END_GET
END_PROPERTY

END_INTERFACE

// 21 Interface/IO_SLOT/ITF_IO_SLOT
INTERFACE ITF_IO_SLOT EXTENDS __System.IQueryinterface

{attribute 'estimated-stack-usage' := '104'}
PROPERTY BIG_SYBIL : ITF_IO_SLOT
GET
END_GET
SET
END_SET
END_PROPERTY

{attribute 'estimated-stack-usage' := '104'}
PROPERTY LOW_SYBIL : ITF_IO_SLOT
GET
END_GET
SET
END_SET
END_PROPERTY

PROPERTY SELF : ITF_IO_SLOT
GET
END_GET
END_PROPERTY

PROPERTY PARENT : ITF_IO_DEVICE
SET
END_SET
GET
END_GET
END_PROPERTY

PROPERTY SLOT_NR : USINT
SET
END_SET
GET
END_GET
END_PROPERTY

PROPERTY IMAGE : STRING
GET
END_GET
SET
END_SET
END_PROPERTY

PROPERTY DYN_SIZE : UDINT
GET
END_GET
END_PROPERTY

METHOD GET_IO : ITF_IO
VAR_INPUT
	_usiIoNr			: 	USINT;
END_VAR
END_METHOD

METHOD CREATE_IO : BOOL
VAR_INPUT
	_usiIoNr			: 	USINT;
	_enType				:	enIOType;
END_VAR
END_METHOD

PROPERTY AY_ITF_IO_VIS : ARRAY[1..16] OF ITF_IO;
GET
END_GET
END_PROPERTY

METHOD RELOAD_ARRAY
VAR_INPUT
	xInit		: BOOL;
	xLoadNext16	: BOOL;
	xLoadLast16	: BOOL;
END_VAR
END_METHOD

{attribute 'monitoring' := 'call'}
PROPERTY SELFPOINTER : POINTER TO FB_IO_SLOT
GET
END_GET
END_PROPERTY

PROPERTY COUNT : USINT
GET
END_GET
END_PROPERTY

METHOD CHECK_SLOT : BOOL
VAR_INPUT
	enCheckIoIn		:	enCheckIo;
	usiAnzIoType	:	USINT;
END_VAR
END_METHOD

END_INTERFACE

// 30 Program Organization Units/IO_SLOT/FB_IO_SLOT
{attribute 'enable_dynamic_creation'}
FUNCTION_BLOCK FB_IO_SLOT IMPLEMENTS ITF_IO_SLOT
VAR_INPUT
END_VAR
VAR_OUTPUT
	udiDynMem					:	UDINT;	
END_VAR
VAR
	usiSlotNr					:	USINT;
	
	_IMAGE						:	STRING;
	
	_ITF_PARENT					:	ITF_IO_DEVICE;	

	_ITF_BIG_SYBIL				:	ITF_IO_SLOT;
	_ITF_LOW_SYBIL				:	ITF_IO_SLOT;
	                			
	_BASE_IO					:	ITF_IO;
	_TEMP_REG_IO				:	ITF_IO;
	_NEXT_IO_LAST_GET			:	ITF_IO;	
	
	_COUNT						:	USINT;
	_COUNT_DI					:	USINT;
	_COUNT_AI					:	USINT;
	_COUNT_DO					:	USINT;
	_COUNT_AO					:	USINT;
	_udiDynMemTemp				:	UDINT;	
	_ayITF_IOS					:	ARRAY[1..16] OF ITF_IO;
	_ayITF_IO_VIS				:	ARRAY[1..16] OF ITF_IO;
END_VAR

METHOD ADD_IO
VAR_INPUT
	ITF_IO_IN		:	ITF_IO;
END_VAR
VAR
	ITF_TEMP		:	ITF_IO;
	ITF_TEMP_BIG	:	ITF_IO;
	ITF_TEMP_LOW	:	ITF_IO;
	xDone			:	BOOL;
END_VAR
(* Check if Valid Interface Input *)
IF __QUERYINTERFACE(ITF_IO_IN,ITF_IO_IN) THEN
	ITF_IO_IN.PARENT := THIS^;
	IF TO_DINT(ITF_IO_IN.IO_NR) >= LOWER_BOUND(_ayITF_IOS,1) AND
	   TO_DINT(ITF_IO_IN.IO_NR) <= UPPER_BOUND(_ayITF_IOS,1) THEN
	   _ayITF_IOS[ITF_IO_IN.IO_NR] := ITF_IO_IN;
	END_IF;
	(* Check if Valid Interface Base*)
	IF __QUERYINTERFACE(_BASE_IO,_BASE_IO) THEN
		(* Check if Valid Interface Temporary registration *)
		IF __QUERYINTERFACE(_TEMP_REG_IO,ITF_TEMP) THEN
			REPEAT
				(* Get Big Sybil of registration *)
				IF __QUERYINTERFACE(ITF_TEMP.BIG_SYBIL,ITF_TEMP_BIG) THEN
					(* Check if IO Type is Lower or Bigger *)
					IF ITF_IO_IN.IO_TYPE <= ITF_TEMP.IO_TYPE AND
						ITF_IO_IN.IO_TYPE >= ITF_TEMP_BIG.IO_TYPE THEN
						(* Check if Adress is Lower *)
						IF ITF_IO_IN.IO_NR <= ITF_TEMP.IO_NR THEN
							(* Check if Adress is Bigger and update if yes*)
							IF ITF_IO_IN.IO_NR >= ITF_TEMP_BIG.IO_NR THEN
								ITF_IO_IN.BIG_SYBIL := ITF_TEMP.BIG_SYBIL;
								ITF_IO_IN.LOW_SYBIL := ITF_TEMP;
								xDone	 := TRUE;							
							END_IF;
						(* Adress is Bigger update *)
						ELSE
							IF __QUERYINTERFACE(ITF_TEMP.LOW_SYBIL,ITF_TEMP_LOW) THEN
								IF ITF_IO_IN.IO_TYPE < ITF_TEMP_LOW.IO_TYPE OR
									(ITF_IO_IN.IO_TYPE = ITF_TEMP_LOW.IO_TYPE AND
									ITF_IO_IN.IO_NR <= ITF_TEMP_LOW.IO_NR) THEN
									ITF_IO_IN.LOW_SYBIL := ITF_TEMP.LOW_SYBIL;
									ITF_IO_IN.BIG_SYBIL := ITF_TEMP;
									xDone	 := TRUE;
								END_IF;
							ELSE
								ITF_IO_IN.LOW_SYBIL := ITF_TEMP.LOW_SYBIL;
								ITF_IO_IN.BIG_SYBIL := ITF_TEMP;
								xDone	 := TRUE;
								(* Update Registation Job if temp is the last one *)
								IF ITF_TEMP = _TEMP_REG_IO THEN
									_TEMP_REG_IO := ITF_IO_IN;
									_TEMP_REG_IO.LOW_SYBIL := 0;
								END_IF;
							END_IF;
						END_IF;
					(* Function Code ist Bigger Insert after temporary*)
					ELSIF ITF_IO_IN.IO_TYPE > ITF_TEMP.IO_TYPE THEN
						ITF_IO_IN.LOW_SYBIL := ITF_TEMP.LOW_SYBIL;
						ITF_IO_IN.BIG_SYBIL := ITF_TEMP;
						xDone	 := TRUE;
						(* Update Registation Job if temp is the last one *)
						IF ITF_TEMP = _TEMP_REG_IO THEN
							_TEMP_REG_IO := ITF_IO_IN;
							_TEMP_REG_IO.LOW_SYBIL := 0;
						END_IF
					END_IF;
				(* Interface is same as the Base*)
				ELSIF ITF_TEMP = _BASE_IO THEN
					(* Check if the Input Interface needs to be the new base*)
					IF ITF_IO_IN.IO_NR <= ITF_TEMP.IO_NR THEN 
						ITF_IO_IN.LOW_SYBIL := ITF_TEMP;
						_BASE_IO 			:= ITF_IO_IN;
						_BASE_IO.BIG_SYBIL 	:= 0;
						xDone	 			:= TRUE; 
					ELSE
						(* Update Registation Job if temp is the last one *)
						IF ITF_TEMP = _TEMP_REG_IO THEN
							_TEMP_REG_IO			:= ITF_IO_IN;
							_TEMP_REG_IO.LOW_SYBIL 	:= 0;
						END_IF
						ITF_IO_IN.LOW_SYBIL := _BASE_IO.LOW_SYBIL;
						_BASE_IO.LOW_SYBIL 	:= ITF_IO_IN;
					END_IF;
				END_IF;
				(* Get Next Interface to Check*)
				__QUERYINTERFACE(ITF_TEMP.BIG_SYBIL,ITF_TEMP);
			UNTIL xDone OR ITF_TEMP = 0 
			END_REPEAT
		ELSE
			(* Set Base Low sybill on second call*)
			_BASE_IO.LOW_SYBIL 	:= ITF_IO_IN;
			_TEMP_REG_IO 		:= ITF_IO_IN;		
		END_IF;		
	ELSE
		(* Set Base on first call*)
		_BASE_IO 		:= ITF_IO_IN;
		_TEMP_REG_IO 	:= ITF_IO_IN;
	END_IF;
	(* Count Jobs *)
	_COUNT := _COUNT + 1;
	THIS^.RELOAD_ARRAY(TRUE,FALSE,FALSE);
END_IF;
END_METHOD

METHOD CHECK_IF_IO_EXIST : BOOL
VAR_INPUT
	_usiIoNr			: 	USINT;
	_enType				:	enIOType;
END_VAR
VAR
	_TEMP_CHK_IO	:	ITF_IO;
	udiSafe			:	UDINT;
END_VAR
IF __QUERYINTERFACE(_BASE_IO,_TEMP_CHK_IO) THEN
	REPEAT 
		IF _TEMP_CHK_IO.IO_NR = _usiIoNr AND
			_TEMP_CHK_IO.IO_TYPE	= _enType THEN
			CHECK_IF_IO_EXIST := TRUE;
		END_IF;
		_TEMP_CHK_IO := _TEMP_CHK_IO.LOW_SYBIL;
		udiSafe	:= udiSafe + 1;
	UNTIL CHECK_IF_IO_EXIST OR _TEMP_CHK_IO = 0 OR udiSafe >= 16#FFFFFFFE
	END_REPEAT
ELSE
	CHECK_IF_IO_EXIST := FALSE;
END_IF
END_METHOD

METHOD CREATE_IO : BOOL
VAR_INPUT
	_usiIoNr			: 	USINT;
	_enType				:	enIOType;
END_VAR
VAR	
	pFbDI				:	POINTER TO FB_DI;
	pFbDO				:	POINTER TO FB_DO;
	pFbAI				:	POINTER TO FB_AI;
	pFbAO				:	POINTER TO FB_AO;
END_VAR
IF NOT CHECK_IF_IO_EXIST(_usiIoNr,_enType) THEN
	IF _enType = enIOType.Digital_IN THEN
		pFbDI := __NEW(FB_DI);
		IF pFbDI <> 0 THEN
			_udiDynMemTemp	:= _udiDynMemTemp + SIZEOF(FB_DI);		
			pFbDI^.IO_NR	:= _usiIoNr;
			pFbDI^.SLOT_NR	:= usiSlotNr;
			pFbDI^.IO_TYPE	:= _enType;
		
			IF __QUERYINTERFACE(_ITF_PARENT,_ITF_PARENT) THEN
				pFbDI^.ProSetInstancePathOnDynCreate 	:= 	Standard.CONCAT(
															Standard.CONCAT(
															Standard.CONCAT(
															Standard.CONCAT(
															Standard.CONCAT(
															Standard.CONCAT(
															Standard.CONCAT(
															Standard.CONCAT(_ITF_PARENT.INSTANCE_PATH,
																			'.SLOT_'),
																			TO_STRING(SLOT_NR)),
																			'.'),
																			TO_STRING(_enType)),
																			'_'),
																			TO_STRING(_usiIoNr)),
																			'.'),
																			'FbConfigFile');														
				ADD_IO(pFbDI^);
				_ITF_PARENT.ADDITION_DYN_SIZE := + SIZEOF(FB_DI);
				_COUNT_DI := _COUNT_DI + 1;
			ELSE
				pFbDI^.DESTROY();
			END_IF;
		ELSE
			ADD_ERROR();
		END_IF;		
		
	ELSIF _enType = enIOType.Digital_OUT THEN
		pFbDO := __NEW(FB_DO);
		IF pFbDO <> 0 THEN
			_udiDynMemTemp	:= _udiDynMemTemp + SIZEOF(FB_DO);		
			pFbDO^.IO_NR	:= _usiIoNr;
			pFbDO^.SLOT_NR	:= usiSlotNr;
			pFbDO^.IO_TYPE	:= _enType;
		
			IF __QUERYINTERFACE(_ITF_PARENT,_ITF_PARENT) THEN
				pFbDO^.ProSetInstancePathOnDynCreate 	:= 	Standard.CONCAT(
															Standard.CONCAT(
															Standard.CONCAT(
															Standard.CONCAT(
															Standard.CONCAT(
															Standard.CONCAT(
															Standard.CONCAT(
															Standard.CONCAT(_ITF_PARENT.INSTANCE_PATH,
																			'.SLOT_'),
																			TO_STRING(SLOT_NR)),
																			'.'),
																			TO_STRING(_enType)),
																			'_'),
																			TO_STRING(_usiIoNr)),
																			'.'),
																			'FbConfigFile');		
				ADD_IO(pFbDO^);
				_ITF_PARENT.ADDITION_DYN_SIZE := + SIZEOF(FB_DO);
				_COUNT_DO := _COUNT_DO + 1;
			ELSE
				pFbDO^.DESTROY();
			END_IF;
		ELSE
			ADD_ERROR();
		END_IF;	
		
	ELSIF _enType = enIOType.DC_0_10V_IN OR  
		  _enType = enIOType.DC_0_20mA_IN OR 
		  _enType = enIOType.DC_4_20mA_IN OR
		  _enType = enIOType.TEMPERATUR	OR 
		  _enType = enIOType.OHM THEN
		pFbAI := __NEW(FB_AI);
		IF pFbAI <> 0 THEN
			_udiDynMemTemp	:= _udiDynMemTemp + SIZEOF(FB_AI);		
			pFbAI^.IO_NR	:= _usiIoNr;
			pFbAI^.SLOT_NR	:= usiSlotNr;
			pFbAI^.IO_TYPE	:= _enType;
		
			IF __QUERYINTERFACE(_ITF_PARENT,_ITF_PARENT) THEN
				pFbAI^.ProSetInstancePathOnDynCreate 	:= 	Standard.CONCAT(
															Standard.CONCAT(
															Standard.CONCAT(
															Standard.CONCAT(
															Standard.CONCAT(
															Standard.CONCAT(
															Standard.CONCAT(
															Standard.CONCAT(_ITF_PARENT.INSTANCE_PATH,
																			'.SLOT_'),
																			TO_STRING(SLOT_NR)),
																			'.'),
																			TO_STRING(_enType)),
																			'_'),
																			TO_STRING(_usiIoNr)),
																			'.'),
																			'FbConfigFile');																	
				ADD_IO(pFbAI^);
				_ITF_PARENT.ADDITION_DYN_SIZE := + SIZEOF(FB_AI);
				_COUNT_AI := _COUNT_AI + 1;
			ELSE
				pFbAI^.DESTROY();
			END_IF;
		ELSE
			ADD_ERROR();
		END_IF;	
	ELSIF _enType = enIOType.DC_0_10V_OUT OR  
		  _enType = enIOType.DC_0_20mA_OUT OR 
		  _enType = enIOType.DC_4_20mA_OUT THEN
		pFbAO := __NEW(FB_AO);
		IF pFbAO <> 0 THEN
			_udiDynMemTemp	:= _udiDynMemTemp + SIZEOF(FB_AO);		
			pFbAO^.IO_NR	:= _usiIoNr;
			pFbAO^.SLOT_NR	:= usiSlotNr;
			pFbAO^.IO_TYPE	:= _enType;
		
			IF __QUERYINTERFACE(_ITF_PARENT,_ITF_PARENT) THEN
				pFbAO^.ProSetInstancePathOnDynCreate 	:= 	Standard.CONCAT(
															Standard.CONCAT(
															Standard.CONCAT(
															Standard.CONCAT(
															Standard.CONCAT(
															Standard.CONCAT(
															Standard.CONCAT(
															Standard.CONCAT(_ITF_PARENT.INSTANCE_PATH,
																			'.SLOT_'),
																			TO_STRING(SLOT_NR)),
																			'.'),
																			TO_STRING(_enType)),
																			'_'),
																			TO_STRING(_usiIoNr)),
																			'.'),
																			'FbConfigFile');	
				ADD_IO(pFbAO^);
				_ITF_PARENT.ADDITION_DYN_SIZE := + SIZEOF(FB_AO);
				_COUNT_AO := _COUNT_AO + 1;
			ELSE
				pFbAO^.DESTROY();
			END_IF;
		ELSE
			ADD_ERROR();
		END_IF;	
	END_IF;	
	udiDynMem								:= MAX(udiDynMem,_udiDynMemTemp);
END_IF;
END_METHOD

METHOD GET_IO : ITF_IO
VAR_INPUT
	_usiIoNr			: 	USINT;
END_VAR
VAR
	_TEMP_GET_IO	:	ITF_IO;
	udiSafe			:	UDINT;
	xNextIoInUse	:	BOOL;
END_VAR
IF TO_DINT(_usiIoNr) >= LOWER_BOUND(_ayITF_IOS,1) AND
   TO_DINT(_usiIoNr) <= UPPER_BOUND(_ayITF_IOS,1) THEN
   GET_IO := _ayITF_IOS[_usiIoNr];
END_IF;
IF GET_IO = 0 THEN
	IF __QUERYINTERFACE(_NEXT_IO_LAST_GET,_TEMP_GET_IO) THEN
		xNextIoInUse := TRUE;
	ELSIF __QUERYINTERFACE(_BASE_IO,_TEMP_GET_IO) THEN
		xNextIoInUse := FALSE;
	END_IF;
	
	IF __QUERYINTERFACE(_TEMP_GET_IO,_TEMP_GET_IO) THEN
		REPEAT 
			IF _TEMP_GET_IO.IO_NR = _usiIoNr THEN
				GET_IO := _TEMP_GET_IO;
			END_IF;
			_TEMP_GET_IO := _TEMP_GET_IO.LOW_SYBIL;
			_NEXT_IO_LAST_GET := _TEMP_GET_IO;
			IF _TEMP_GET_IO = 0 AND xNextIoInUse THEN
				__QUERYINTERFACE(_BASE_IO,_TEMP_GET_IO);
				xNextIoInUse := FALSE;
			END_IF;
			udiSafe	:= udiSafe + 1;
		UNTIL GET_IO <> 0 OR _TEMP_GET_IO = 0 OR udiSafe >= 16#FFFFFFFE
		END_REPEAT
	ELSE
		GET_IO := 0;
	END_IF;
END_IF;
END_METHOD

{attribute 'estimated-stack-usage' := '104'}
PROPERTY BIG_SYBIL : ITF_IO_SLOT
GET
BIG_SYBIL := _ITF_BIG_SYBIL;
END_GET
SET
_ITF_BIG_SYBIL := BIG_SYBIL;
IF __QUERYINTERFACE(_ITF_BIG_SYBIL,_ITF_BIG_SYBIL) THEN
	IF _ITF_BIG_SYBIL.LOW_SYBIL <> SELF THEN
		_ITF_BIG_SYBIL.LOW_SYBIL := THIS^;
	END_IF;
END_IF;
END_SET
END_PROPERTY

{attribute 'estimated-stack-usage' := '104'}
PROPERTY LOW_SYBIL : ITF_IO_SLOT
GET
LOW_SYBIL := _ITF_LOW_SYBIL;
END_GET
SET
_ITF_LOW_SYBIL := LOW_SYBIL;
IF __QUERYINTERFACE(_ITF_LOW_SYBIL,_ITF_LOW_SYBIL) THEN
	IF _ITF_LOW_SYBIL.BIG_SYBIL <> SELF THEN
		_ITF_LOW_SYBIL.BIG_SYBIL := THIS^;
	END_IF;
END_IF;
END_SET
END_PROPERTY

PROPERTY PARENT : ITF_IO_DEVICE
GET
PARENT := _ITF_PARENT;
END_GET
SET
_ITF_PARENT := PARENT;
END_SET
END_PROPERTY

PROPERTY SELF : ITF_IO_SLOT
GET
SELF := THIS^;
END_GET
END_PROPERTY

PROPERTY SLOT_NR : USINT
GET
SLOT_NR := usiSlotNr;
END_GET
SET
usiSlotNr := SLOT_NR;
END_SET
END_PROPERTY

PROPERTY IMAGE : STRING
GET
IMAGE := _IMAGE;
END_GET
SET
_IMAGE := IMAGE;
END_SET
END_PROPERTY

PROPERTY DYN_SIZE : UDINT
GET
DYN_SIZE := udiDynMem;
END_GET
END_PROPERTY

METHOD RELOAD_ARRAY
VAR_INPUT
	xInit	: BOOL;
	xLoadNext16	: BOOL;
	xLoadLast16	: BOOL;
END_VAR
VAR
	diFor				:	DINT;
	ITF_TEMP_CLIENT_VIS	:	ITF_IO;
	ITF_TEMP_SAFE		:	ITF_IO;
	ITF_TEMP_LAST_VALID	:	ITF_IO;
END_VAR
(* Init Array *)
IF xInit THEN
	_ayITF_IO_VIS[LOWER_BOUND(_ayITF_IO_VIS,1)] := _BASE_IO;
	FOR diFor := LOWER_BOUND(_ayITF_IO_VIS,1) TO UPPER_BOUND(_ayITF_IO_VIS,1) -1 DO
		IF __QUERYINTERFACE(_ayITF_IO_VIS[diFor],ITF_TEMP_CLIENT_VIS) THEN
			_ayITF_IO_VIS[diFor + 1]	:= _ayITF_IO_VIS[diFor].LOW_SYBIL;
		ELSE
			_ayITF_IO_VIS[diFor + 1] := 0;
		END_IF;	
	END_FOR;
(* Load Next 16 *)
ELSIF xLoadNext16 THEN
	IF __QUERYINTERFACE(_ayITF_IO_VIS[UPPER_BOUND(_ayITF_IO_VIS,1)],ITF_TEMP_CLIENT_VIS) THEN
		_ayITF_IO_VIS[LOWER_BOUND(_ayITF_IO_VIS,1)] := ITF_TEMP_CLIENT_VIS.LOW_SYBIL;
		FOR diFor := LOWER_BOUND(_ayITF_IO_VIS,1) TO UPPER_BOUND(_ayITF_IO_VIS,1) -1 DO
			IF __QUERYINTERFACE(_ayITF_IO_VIS[diFor],ITF_TEMP_CLIENT_VIS) THEN
				_ayITF_IO_VIS[diFor + 1]	:= _ayITF_IO_VIS[diFor].LOW_SYBIL;
			ELSE
				_ayITF_IO_VIS[diFor + 1] := 0;
			END_IF;	
		END_FOR;
	END_IF;
(* Load Last 16 *)
ELSIF xLoadLast16 THEN
	IF __QUERYINTERFACE(_ayITF_IO_VIS[LOWER_BOUND(_ayITF_IO_VIS,1)],ITF_TEMP_CLIENT_VIS) THEN
		IF __QUERYINTERFACE(_ayITF_IO_VIS[LOWER_BOUND(_ayITF_IO_VIS,1)].BIG_SYBIL,ITF_TEMP_SAFE) THEN
			_ayITF_IO_VIS[UPPER_BOUND(_ayITF_IO_VIS,1)] := ITF_TEMP_CLIENT_VIS.BIG_SYBIL;
			FOR diFor := UPPER_BOUND(_ayITF_IO_VIS,1) TO LOWER_BOUND(_ayITF_IO_VIS,1) + 1 BY -1 DO 
				IF __QUERYINTERFACE(_ayITF_IO_VIS[diFor],ITF_TEMP_CLIENT_VIS) THEN
					ITF_TEMP_LAST_VALID  			:= _ayITF_IO_VIS[diFor];
					_ayITF_IO_VIS[diFor - 1]	:= _ayITF_IO_VIS[diFor].BIG_SYBIL;
				ELSE
					(* Resort if new ones Inside *)
					_ayITF_IO_VIS[LOWER_BOUND(_ayITF_IO_VIS,1)] := ITF_TEMP_LAST_VALID;
					FOR diFor := LOWER_BOUND(_ayITF_IO_VIS,1) TO UPPER_BOUND(_ayITF_IO_VIS,1) -1 DO
						IF __QUERYINTERFACE(_ayITF_IO_VIS[diFor],ITF_TEMP_CLIENT_VIS) THEN
							_ayITF_IO_VIS[diFor + 1]	:= _ayITF_IO_VIS[diFor].LOW_SYBIL;
						ELSE
							_ayITF_IO_VIS[diFor + 1] := 0;
						END_IF;	
					END_FOR;					
				END_IF;	
			END_FOR;
		END_IF;
	END_IF;	
END_IF;
END_METHOD

PROPERTY AY_ITF_IO_VIS : ARRAY[1..16] OF ITF_IO;
GET
AY_ITF_IO_VIS := _ayITF_IO_VIS;
END_GET
END_PROPERTY

{attribute 'monitoring' := 'call'}
PROPERTY SELFPOINTER : POINTER TO FB_IO_SLOT
GET
SELFPOINTER := THIS;
END_GET
END_PROPERTY

PROPERTY COUNT : USINT
GET
COUNT := _COUNT;
END_GET
END_PROPERTY

METHOD ADD_ERROR
VAR_INPUT
END_VAR
VAR
	ITF_IO_DEVICE_TEMP	:	ITF_IO_DEVICE;
END_VAR
IF __QUERYINTERFACE(_ITF_PARENT,_ITF_PARENT) THEN
	ITF_IO_DEVICE_TEMP.ADD_ERROR();
END_IF;
END_METHOD

METHOD CHECK_SLOT : BOOL
VAR_INPUT
	enCheckIoIn		:	enCheckIo;
	usiAnzIoType	:	USINT;
END_VAR
IF enCheckIoIn = enCheckIo.DI_IO THEN
	IF usiAnzIoType = _COUNT_DI THEN
		CHECK_SLOT := TRUE;
	ELSE
		CHECK_SLOT := FALSE;
	END_IF;
ELSIF enCheckIoIn = enCheckIo.AI_IO THEN
	IF usiAnzIoType = _COUNT_AI THEN
		CHECK_SLOT := TRUE;
	ELSE
		CHECK_SLOT := FALSE;
	END_IF;
ELSIF enCheckIoIn = enCheckIo.DO_IO THEN
	IF usiAnzIoType = _COUNT_DO THEN
		CHECK_SLOT := TRUE;
	ELSE
		CHECK_SLOT := FALSE;
	END_IF;
ELSIF enCheckIoIn = enCheckIo.AO_IO THEN
	IF usiAnzIoType = _COUNT_AO THEN
		CHECK_SLOT := TRUE;
	ELSE
		CHECK_SLOT := FALSE;
	END_IF;
END_IF;
END_METHOD

END_FUNCTION_BLOCK

// 30 Program Organization Units/IO_FB/DI/FB_DI
{attribute 'enable_dynamic_creation'}
FUNCTION_BLOCK FB_DI EXTENDS FB_IO IMPLEMENTS ITF_DI
VAR_INPUT
END_VAR
VAR_OUTPUT
END_VAR
VAR
	// Channel input
	xChannelIn						: BOOL;
	
	// Übergabe variablen
	xValue							: BOOL;
	(* Trendlog *)
	fbTrendLogxValue				: CtaAppInfluxLog.FB_LOG_NODE_BOOL;	
	(*Parameter*)
	fbxInvert						: CtaSysConfig.fbBOOL;
	fbxSimulationValue				: CtaSysConfig.fbBOOL;
END_VAR

METHOD metConfig
VAR_INPUT
END_VAR
fbConfigFile();

fbxSimulation 					(_usiParaNr := 1, itfConfigFb := fbConfigFile);
fbxSimulationLock				(_usiParaNr := 2, itfConfigFb := fbConfigFile);
fbxInvert						(_usiParaNr := 3, itfConfigFb := fbConfigFile);
fbxSimulationValue				(_usiParaNr := 4, itfConfigFb := fbConfigFile);
END_METHOD

PROPERTY proPhysikalValueVisu : String(6)
GET
// Schreiben des physikalischen Wertes für Visualisierung 
proPhysikalValueVisu := TO_STRING(proValue);
END_GET
END_PROPERTY

METHOD FINAL metCyclicIoUpdate
VAR_INPUT
	_xChannelIn : BOOL;
	_xOk		: BOOL;
END_VAR
(* Config *)
metConfig();

(* Chanel Value *)
xChannelIn	:= _xChannelIn;
xOK 		:= _xOk;
// Bei aktivierter Simulation wird der Simulationswert übertragen
IF fbxSimulation.xValue AND NOT fbxSimulationLock.xValue THEN
	xValue := fbxSimulationValue.xValue;
	(* ADD HAND Message *)
	ADD_HAND();
ELSE
	(* REM HAND Message *)
	REM_HAND();
	xValue := xChannelIn;
	fbxSimulationValue.metNewValueNoSave(xChannelIn);
END_IF
(* TREND *)
metTrendLog();
END_METHOD

METHOD metTrendLog
IF NOT fbTrendLogxValue.ENABLE THEN
	fbTrendLogxValue.ENABLE := TRUE;
	fbTrendLogxValue.KEY	:= proLogName;
END_IF;
fbTrendLogxValue.SET_VALUE	:= xChannelIn;
END_METHOD

PROPERTY P_scfbDI_fbxSimulationValue : CtaSysConfig.ITF_DATATYPE
GET
P_scfbDI_fbxSimulationValue := fbxSimulationValue;
END_GET
END_PROPERTY

PROPERTY P_scfbDI_fbxInvert : CtaSysConfig.ITF_DATATYPE
GET
P_scfbDI_fbxInvert := fbxInvert;
END_GET
END_PROPERTY

PROPERTY P_All_Init : scDI_Para
SET
fbxSimulationLock._WertInit := P_All_Init.xSimulationLock;
fbxInvert._WertInit 		:= P_All_Init.xInvert;
END_SET
END_PROPERTY

PROPERTY proValue : BOOL
GET
// Invertierung des Wertes bei aktiver Invertierung
proValue := xValue XOR fbxInvert.proValue;
END_GET
END_PROPERTY

PROPERTY proIsBOOL_IO : BOOL
GET
proIsBOOL_IO := TRUE;
END_GET
END_PROPERTY

END_FUNCTION_BLOCK

// 30 Program Organization Units/IO_FB/IO/FB_IO
{attribute 'enable_dynamic_creation'}
FUNCTION_BLOCK FB_IO EXTENDS FB_IO_TABLE IMPLEMENTS ITF_IO
VAR_INPUT
END_VAR
VAR_OUTPUT
END_VAR
VAR
	(* IO *)
	usiIoNr				: 	USINT;
	usiSlotNr			: 	USINT;
	enType				:	enIOType;
	xOK					: 	BOOL;
	xIoSim				:	BOOL;
	xTrigError			:	BOOL;
	xTrigHand			:	BOOL;
	(* ITF *)
	_ITF_BIG_SYBIL		:	ITF_IO;
	_ITF_LOW_SYBIL		:	ITF_IO;
	_ITF_PARENT			:	ITF_IO_SLOT;
	
	(*Parameter*)
	fbConfigFile		: 	CtaSysConfig.fbConfigFile;

	fbxSimulation		:	CtaSysConfig.fbBOOL;
	fbxSimulationLock	:	CtaSysConfig.fbBOOL;		
END_VAR

PROPERTY SELF : ITF_IO
GET
SELF := THIS^;
END_GET
END_PROPERTY

PROPERTY P_scfbIO_fbxSimulationLock : CtaSysConfig.ITF_DATATYPE
GET
P_scfbIO_fbxSimulationLock := fbxSimulationLock;
END_GET
END_PROPERTY

PROPERTY P_scfbIO_Simulation : CtaSysConfig.ITF_DATATYPE
GET
P_scfbIO_Simulation := fbxSimulation;
END_GET
END_PROPERTY

PROPERTY ProSetInstancePathOnDynCreate : STRING(255)
SET
fbConfigFile.ProSetInstancePathOnDynCreate := ProSetInstancePathOnDynCreate;
END_SET
END_PROPERTY

{attribute 'monitoring' := 'call'}
PROPERTY SELFPOINTER : POINTER TO FB_IO
GET
SELFPOINTER := THIS;
END_GET
END_PROPERTY

PROPERTY IO_TYPE : enIOType
SET
enType := IO_TYPE;
END_SET
GET
IO_TYPE := enType;
END_GET
END_PROPERTY

PROPERTY IO_NR : USINT
GET
IO_NR := usiIoNr;
END_GET
SET
usiIoNr := IO_NR;
END_SET
END_PROPERTY

PROPERTY PARENT : ITF_IO_SLOT
GET
PARENT := _ITF_PARENT;
END_GET
SET
_ITF_PARENT := PARENT;
END_SET
END_PROPERTY

PROPERTY proSimVisu : STRING
GET
// Simbolausgabe für Visu bei aktiver Simulations- Sperre
IF fbxSimulationLock.proValue THEN	
	proSimVisu := 'CtaVisSymbols.ImagePool.lock_closed_black';	
ELSE	
	IF fbxSimulation.proValue THEN
		proSimVisu := 'CtaVisSymbols.ImagePool.front_hand_Yellow';
	ELSE
		proSimVisu := 'CtaVisSymbols.ImagePool.front_hand_Black';
	END_IF	
END_IF
END_GET
END_PROPERTY

PROPERTY proOK : BOOL
GET
// Setzen des Modul OKs 
IF xOK THEN
	proOK := TRUE;
ELSIF xIoSim THEN
	proOK := TRUE;
ELSE
	proOK := FALSE;
END_IF
END_GET
END_PROPERTY

PROPERTY proOkVisu : STRING
GET
// Definition des anzuzeigenden Bildes für Visu
IF xOK THEN
	proOkVisu := 'CtaVisSymbols.ImagePool.check_green';
ELSIF xIoSim THEN
	proOkVisu := 'CtaVisSymbols.ImagePool.front_hand_Yellow';
ELSE
	proOkVisu := 'CtaVisSymbols.ImagePool.CtaError';
END_IF
END_GET
END_PROPERTY

PROPERTY proPhysikalValueVisu : STRING(6)
GET
END_GET
SET
END_SET
END_PROPERTY

PROPERTY proIsSimLocked : BOOL
GET
proIsSimLocked := fbxSimulationLock.proValue;
END_GET
END_PROPERTY

PROPERTY proIsBOOL_IO : BOOL
GET
proIsBOOL_IO := FALSE;
END_GET
END_PROPERTY

METHOD ADD_HAND
VAR_INPUT
END_VAR
VAR
	ITF_IO_DEVICE_TEMP	:	ITF_IO_DEVICE;
END_VAR
IF NOT xTrigHand THEN
	IF __QUERYINTERFACE(_ITF_PARENT,_ITF_PARENT) THEN
		IF __QUERYINTERFACE(_ITF_PARENT.PARENT,ITF_IO_DEVICE_TEMP) THEN
			ITF_IO_DEVICE_TEMP.ADD_HAND();
		END_IF;	
	END_IF;
	xTrigHand := TRUE;
END_IF;
END_METHOD

PROPERTY proLogName : STRING(100)
GET
VAR
	ITF_IO_DEVICE_TEMP	:	ITF_IO_DEVICE;
END_VAR
IF __QUERYINTERFACE(_ITF_PARENT,_ITF_PARENT) THEN
	IF __QUERYINTERFACE(_ITF_PARENT.PARENT,ITF_IO_DEVICE_TEMP) THEN
		proLogName := CONCAT(TO_STRING(_ITF_PARENT.PARENT.DEV_NR),CONCAT('SLOT_',CONCAT(TO_STRING(_ITF_PARENT.SLOT_NR),CONCAT('_DI_',TO_STRING(usiIoNr)))));
	END_IF;
END_IF;
END_GET
END_PROPERTY

METHOD DESTROY
VAR
	pSelf					:	POINTER TO FB_IO;
	ITF_IO_DEVICE_TEMP		:	ITF_IO_DEVICE;
END_VAR
IF __QUERYINTERFACE(_ITF_BIG_SYBIL,_ITF_BIG_SYBIL) THEN
	_ITF_BIG_SYBIL.LOW_SYBIL := _ITF_LOW_SYBIL;
END_IF;

IF __QUERYINTERFACE(_ITF_LOW_SYBIL,_ITF_LOW_SYBIL) THEN
	_ITF_LOW_SYBIL.BIG_SYBIL := _ITF_BIG_SYBIL;
END_IF;

IF __QUERYINTERFACE(_ITF_PARENT,_ITF_PARENT) THEN
	IF __QUERYINTERFACE(_ITF_PARENT.PARENT,ITF_IO_DEVICE_TEMP) THEN
		IF enType = enIOType.Digital_IN 		THEN
			ITF_IO_DEVICE_TEMP.ADDITION_DYN_SIZE := TO_DINT(0 - SIZEOF(FB_DI));
			
		ELSIF enType = enIOType.Digital_OUT 	THEN
			ITF_IO_DEVICE_TEMP.ADDITION_DYN_SIZE := TO_DINT(0 - SIZEOF(FB_DO));

		ELSIF enType = enIOType.DC_0_10V_IN 	OR  
			  enType = enIOType.DC_0_20mA_IN 	OR 
			  enType = enIOType.DC_4_20mA_IN	OR
			  enType = enIOType.TEMPERATUR		OR 
			  enType = enIOType.OHM 			THEN	
			ITF_IO_DEVICE_TEMP.ADDITION_DYN_SIZE := TO_DINT(0 - SIZEOF(FB_AI));
			
		ELSIF enType = enIOType.DC_0_10V_OUT 	OR  
			  enType = enIOType.DC_0_20mA_OUT	OR 
			  enType = enIOType.DC_4_20mA_OUT 	THEN		
			ITF_IO_DEVICE_TEMP.ADDITION_DYN_SIZE := TO_DINT(0 - SIZEOF(FB_AO));		
			
		END_IF;
	END_IF;
END_IF;

pSelf := THIS;

__DELETE(pSelf);
END_METHOD

{attribute 'estimated-stack-usage' := '104'}
PROPERTY BIG_SYBIL : ITF_IO
GET
BIG_SYBIL := _ITF_BIG_SYBIL;
END_GET
SET
_ITF_BIG_SYBIL := BIG_SYBIL;
IF __QUERYINTERFACE(_ITF_BIG_SYBIL,_ITF_BIG_SYBIL) THEN
	IF _ITF_BIG_SYBIL.LOW_SYBIL <> SELF THEN
		_ITF_BIG_SYBIL.LOW_SYBIL := THIS^;
	END_IF;
END_IF;
END_SET
END_PROPERTY

{attribute 'estimated-stack-usage' := '104'}
PROPERTY LOW_SYBIL : ITF_IO
GET
LOW_SYBIL := _ITF_LOW_SYBIL;
END_GET
SET
_ITF_LOW_SYBIL := LOW_SYBIL;
IF __QUERYINTERFACE(_ITF_LOW_SYBIL,_ITF_LOW_SYBIL) THEN
	IF _ITF_LOW_SYBIL.BIG_SYBIL <> SELF THEN
		_ITF_LOW_SYBIL.BIG_SYBIL := THIS^;
	END_IF;
END_IF;
END_SET
END_PROPERTY

PROPERTY SLOT_NR : USINT
GET
SLOT_NR := usiSlotNr;
END_GET
SET
usiSlotNr := SLOT_NR;
END_SET
END_PROPERTY

METHOD REM_HAND
VAR_INPUT
END_VAR
VAR
	ITF_IO_DEVICE_TEMP	:	ITF_IO_DEVICE;
END_VAR
IF xTrigHand THEN
	IF __QUERYINTERFACE(_ITF_PARENT,_ITF_PARENT) THEN
		IF __QUERYINTERFACE(_ITF_PARENT.PARENT,ITF_IO_DEVICE_TEMP) THEN
			ITF_IO_DEVICE_TEMP.REM_HAND();
		END_IF;	
	END_IF;
	xTrigHand := FALSE;
END_IF;
END_METHOD

END_FUNCTION_BLOCK

// 30 Program Organization Units/IO_FB/IO/FB_IO_TABLE
{attribute 'enable_dynamic_creation'}
FUNCTION_BLOCK FB_IO_TABLE IMPLEMENTS ITF_IO_TABLE
VAR_INPUT
END_VAR
VAR_OUTPUT
END_VAR
VAR

END_VAR


PROPERTY IO_NR : USINT
GET
END_GET
SET
END_SET
END_PROPERTY


PROPERTY IO_TYPE : enIOType
GET
END_GET
SET
END_SET
END_PROPERTY


PROPERTY proSimVisu : STRING
GET
END_GET
END_PROPERTY

PROPERTY SLOT_NR : USINT
GET
END_GET
SET
END_SET
END_PROPERTY


PROPERTY proOkVisu : STRING
GET
END_GET
END_PROPERTY


PROPERTY proPhysikalValueVisu : STRING(6)
GET
END_GET
SET
END_SET
END_PROPERTY

END_FUNCTION_BLOCK

// 30 Program Organization Units/IO_FB/DO/FB_DO
{attribute 'enable_dynamic_creation'}
FUNCTION_BLOCK FB_DO EXTENDS FB_IO IMPLEMENTS ITF_DO
VAR_INPUT
END_VAR
VAR_OUTPUT
END_VAR
VAR
	// Value in
	xValueIn	:	BOOL;
	
	// Transfer variable	
	xValue		:	BOOL;
		
	// Channel output
	xChannelOut	:	BOOL;
	(* Trendlog *)
	fbTrendLogxValue				:	CtaAppInfluxLog.FB_LOG_NODE_BOOL;
	(*Parameter*)
	fbxInvert						:	CtaSysConfig.fbBOOL;
	fbxSimulationValue				:	CtaSysConfig.fbBOOL;
END_VAR

PROPERTY P_scfbDO_fbxInvert : CtaSysConfig.ITF_DATATYPE
GET
P_scfbDO_fbxInvert := fbxInvert;
END_GET
END_PROPERTY

PROPERTY P_All_Init : scDO_Para
SET
fbxSimulationLock._WertInit := P_All_Init.xSimulationLock;
fbxInvert._WertInit 		:= P_All_Init.xInvert;
END_SET
END_PROPERTY

PROPERTY P_scfbDO_fbxSimulationValue : CtaSysConfig.ITF_DATATYPE
GET
P_scfbDO_fbxSimulationValue := fbxSimulationValue;
END_GET
END_PROPERTY

METHOD metConfig
VAR_INPUT
END_VAR
fbConfigFile();

fbxSimulation 					(_usiParaNr := 1, itfConfigFb := fbConfigFile);
fbxSimulationLock				(_usiParaNr := 2, itfConfigFb := fbConfigFile);
fbxInvert						(_usiParaNr := 3, itfConfigFb := fbConfigFile);
fbxSimulationValue				(_usiParaNr := 4, itfConfigFb := fbConfigFile);
END_METHOD

METHOD metTrendLog
IF NOT fbTrendLogxValue.ENABLE THEN
	fbTrendLogxValue.ENABLE := TRUE;
	fbTrendLogxValue.KEY	:= proLogName;
END_IF;
fbTrendLogxValue.SET_VALUE	 := xChannelOut;
END_METHOD

PROPERTY proPhysikalValueVisu : String(6)
GET
// Schreiben des physikalischen Wertes für Visualisierung
proPhysikalValueVisu := TO_STRING(xChannelOut);
END_GET
END_PROPERTY

PROPERTY proIsBOOL_IO : BOOL
GET
proIsBOOL_IO := TRUE;
END_GET
END_PROPERTY

PROPERTY proValue : BOOL
GET
proValue := xValue;
END_GET
SET
xValueIn := proValue;
END_SET
END_PROPERTY

METHOD FINAL metCyclicIoUpdate
VAR_INPUT
	_xOk		: BOOL;
END_VAR
VAR_OUTPUT
	_xChannelOut : BOOL;
END_VAR
(* Config *)
metConfig();
// Bei aktiver Simulation wird Simulationswert dem Ausgang übergeben
IF fbxSimulation.xValue AND NOT fbxSimulationLock.xValue THEN
	xValue 	:= fbxSimulationValue.xValue;
	(* ADD HAND Message *)
	ADD_HAND();
ELSE
	(* REM HAND Message *)
	REM_HAND();
	xValue		:= xValueIn;
	fbxSimulationValue.metNewValueNoSave(xValueIn);
END_IF

IF NOT _xOk AND NOT xIoSim THEN
	// Abschaltung des Ausganges bei Kbus Fehler
	xChannelOut := FALSE XOR fbxInvert.xValue;
ELSE	
	// Invertierung des Wertes bei aktiver Invertierung
	xChannelOut := xValue XOR fbxInvert.xValue;
END_IF

xOK			 := _xOk;
_xChannelOut := xChannelOut;

(* TREND *)
metTrendLog();
END_METHOD

END_FUNCTION_BLOCK

// 21 Interface/IO_FB/DO/ITF_DO
INTERFACE ITF_DO EXTENDS ITF_IO

PROPERTY proValue : BOOL
SET
END_SET
GET
END_GET
END_PROPERTY

METHOD FINAL metCyclicIoUpdate
VAR_INPUT
	_xOk		: BOOL;
END_VAR
VAR_OUTPUT
	_xChannelOut : BOOL;
END_VAR
END_METHOD

PROPERTY P_scfbDO_fbxSimulationValue : CtaSysConfig.ITF_DATATYPE
GET
END_GET
END_PROPERTY

PROPERTY P_All_Init : scDO_Para
SET
END_SET
END_PROPERTY

PROPERTY P_scfbDO_fbxInvert : CtaSysConfig.ITF_DATATYPE
GET
END_GET
END_PROPERTY

END_INTERFACE

// 30 Program Organization Units/IO_FB/AI/FB_AI
{attribute 'enable_dynamic_creation'}
FUNCTION_BLOCK FB_AI EXTENDS FB_IO IMPLEMENTS ITF_AI
VAR_INPUT
END_VAR
VAR_OUTPUT
END_VAR
VAR

	(*Value output*)
	rValue				: 	REAL;
	
	
	(*Calculation Vars*)
	rPhysicalValue		:	REAL;	// Physikalischer Wert
	rUserScale			:	REAL;
	
	(*Alarm*)	
	xAlUeberlauf		:	BOOL;	// Alarm Überlauf
	xAlUnterlauf		:	BOOL;	// Alarm Unterlauf
	(* Trendlog *)
	fbTrendLogrValue	:	CtaAppInfluxLog.FB_LOG_NODE_REAL;		
	(*Parameter*)	
	fbrMin				:	CtaSysConfig.fbREAL;			
	fbrMax				:	CtaSysConfig.fbREAL;		
	fbrMinPhysical		:	CtaSysConfig.fbREAL;
	fbstPhysicalUnit	:	CtaSysConfig.fbSTRING40;			
	fbrPhysicalAlarm	:	CtaSysConfig.fbREAL;			
	fbrSimulationValue	:	CtaSysConfig.fbREAL;
	fbrCorrectionValue	:	CtaSysConfig.fbREAL;	
END_VAR

PROPERTY P_scfbAI_fbstPhysicalUnit : CtaSysConfig.ITF_DATATYPE
GET
P_scfbAI_fbstPhysicalUnit := fbstPhysicalUnit;
END_GET
END_PROPERTY

PROPERTY P_scfbAI_fbrMax : CtaSysConfig.ITF_DATATYPE
GET
P_scfbAI_fbrMax := fbrMax;
END_GET
END_PROPERTY

PROPERTY P_scfbAI_fbrMinPhysical : CtaSysConfig.ITF_DATATYPE
GET
P_scfbAI_fbrMinPhysical:= fbrMinPhysical;
END_GET
END_PROPERTY

PROPERTY P_scfbAI_fbrMin : CtaSysConfig.ITF_DATATYPE
GET
P_scfbAI_fbrMin := fbrMin;
END_GET
END_PROPERTY

PROPERTY P_scfbAI_fbrPhysicalAlarm : CtaSysConfig.ITF_DATATYPE
GET
P_scfbAI_fbrPhysicalAlarm := fbrPhysicalAlarm;
END_GET
END_PROPERTY

PROPERTY P_scfbAI_fbrSimulationValue : CtaSysConfig.ITF_DATATYPE
GET
P_scfbAI_fbrSimulationValue := fbrSimulationValue;
END_GET
END_PROPERTY

PROPERTY P_scfbAI_fbrCorrectionValue : CtaSysConfig.ITF_DATATYPE
GET
P_scfbAI_fbrCorrectionValue := fbrCorrectionValue;
END_GET
END_PROPERTY

PROPERTY P_All_Init : scAI_Para
SET
fbxSimulationLock._WertInit 	:= P_All_Init.xSimulationLock;
fbrMin._WertInit				:= P_All_Init.rMin;
fbrMax._WertInit				:= P_All_Init.rMax;
fbrMinPhysical._WertInit		:= P_All_Init.rMinPhysical;
fbrPhysicalAlarm._WertInit		:= P_All_Init.rPhysicalAlarm;
fbrCorrectionValue._WertInit	:= P_All_Init.rCorrectionValue;
fbstPhysicalUnit._WertInit		:= P_All_Init.stPhysicalUnit;
END_SET
END_PROPERTY

PROPERTY proIsBOOL_IO : BOOL
GET
proIsBOOL_IO := FALSE;
END_GET
END_PROPERTY

PROPERTY proPhysikalValueVisu : STRING(6)
GET
// Schreiben des physikalischen Wertes für Visualisierung
IF FIND(TO_STRING(proPhysicalValue),'.') <> 0 THEN
	proPhysikalValueVisu := LEFT(TO_STRING(proPhysicalValue),(FIND(TO_STRING(proPhysicalValue),'.')+1));	
ELSE
	proPhysikalValueVisu := TO_STRING(proPhysicalValue);
END_IF
END_GET
END_PROPERTY

PROPERTY proPhysicalValue : REAL
GET
// Ausgabe Simulationswert bei aktiver Simulation
IF fbxSimulation.proValue THEN
	proPhysicalValue := fbrSimulationValue.rValue;
ELSE
	proPhysicalValue := rPhysicalValue;
END_IF
END_GET
END_PROPERTY

PROPERTY proValue : REAL
GET
(*Wert mit Korrektur*)
proValue := rValue;
END_GET
END_PROPERTY

METHOD FINAL metCyclicIoUpdate
VAR_INPUT
	_xOk				: BOOL;
	_rPhysicalValue 	: REAL;
	_xAlUeberlauf		: BOOL;
	_xAlUnterlauf		: BOOL;
END_VAR
VAR
	xTempAlUnterlauf	: BOOL;
END_VAR
(* Config *)
metConfig();

// Signalausgabe an PGM, bei aktiver Simulation = Simulationswert
IF NOT fbxSimulation.xValue OR fbxSimulationLock.xValue THEN
		(* Skalieren aller Analogen Inputs welche nicht Ohmisch oder Temperatur sind *)
		IF enType <> enIOType.TEMPERATUR AND enType <> enIOType.OHM THEN
			rUserScale := fcScaleIn(	rValueIn 		:= 	_rPhysicalValue,
										rMin 			:= 	fbrMin.rValue,
										rMax 			:= 	fbrMax.rValue,
										rMinPysical 	:=	fbrMinPhysical.rValue,
										rPysicalAlarm	:=	fbrPhysicalAlarm.rValue,
										enType			:=  enType,
										xAlUnterlauf	=>	xTempAlUnterlauf);
		ELSE
			rUserScale := _rPhysicalValue;	
		END_IF;							
	// Übergabe des skalierten Eingangssignals
	rValue						:= rUserScale  + fbrCorrectionValue.rValue;
	fbrSimulationValue.metNewValueNoSave(proPhysicalValue);  
	(* REM HAND Message *)
	REM_HAND();
	(* Set Scale *)
	CASE enType OF
		enIOType.DC_0_10V_IN,enIOType.DC_0_10V_OUT:
			fbrSimulationValue.metNewMinMax(0,10); 
		enIOType.DC_0_20mA_OUT:
			fbrSimulationValue.metNewMinMax(0,20); 
		enIOType.DC_4_20mA_IN,enIOType.DC_4_20mA_OUT:
			fbrSimulationValue.metNewMinMax(4,20);
		enIOType.TEMPERATUR:
			fbrSimulationValue.metNewMinMax(-2000,8500);
		enIOType.OHM:
			fbrSimulationValue.metNewMinMax(1.0E-44,3.402823E+38);
	END_CASE	
ELSE
	(* ADD HAND Message *)
	ADD_HAND();
	(* Set Scale *)
	CASE enType OF
		enIOType.DC_0_10V_IN,enIOType.DC_0_10V_OUT:
			fbrSimulationValue.metNewMinMax(0,10); 
		enIOType.DC_0_20mA_OUT:
			fbrSimulationValue.metNewMinMax(0,20); 
		enIOType.DC_4_20mA_IN,enIOType.DC_4_20mA_OUT:
			fbrSimulationValue.metNewMinMax(4,20);
		enIOType.TEMPERATUR:
			fbrSimulationValue.metNewMinMax(-2000,8500);
		enIOType.OHM:
			fbrSimulationValue.metNewMinMax(1.0E-44,3.402823E+38);
	END_CASE	
	IF enType = enIOType.TEMPERATUR OR enType = enIOType.OHM THEN
		rValue              := fbrSimulationValue.rValue;   
	ELSE	
		// Skalierung des Simulationswertes
		rValue := fcScaleIn(	rValueIn 		:= 	fbrSimulationValue.rValue,
								rMin 			:= 	fbrMin.rValue,
								rMax 			:= 	fbrMax.rValue,
								rMinPysical 	:=	fbrMinPhysical.rValue,
								rPysicalAlarm	:=	fbrPhysicalAlarm.rValue,
								enType			:=  enType,
								xAlUnterlauf	=>	xTempAlUnterlauf);
									
	END_IF
END_IF

rPhysicalValue	:= _rPhysicalValue;	
(*Alarm*)	        
xAlUeberlauf	:= _xAlUeberlauf;	
xAlUnterlauf 	:= _xAlUnterlauf OR xTempAlUnterlauf;
(* Update Info *)
xOK				:= _xOk AND NOT xAlUeberlauf AND NOT xAlUnterlauf;

(* TREND *)             
metTrendLog();
END_METHOD

METHOD metTrendLog
IF NOT fbTrendLogrValue.ENABLE THEN
	fbTrendLogrValue.ENABLE := TRUE;
	fbTrendLogrValue.KEY	:= proLogName;
END_IF;
fbTrendLogrValue.SET_VALUE	:= rPhysicalValue;
END_METHOD

PROPERTY proAlUeberlauf : BOOL
GET
proAlUeberlauf := xAlUeberlauf;
END_GET
END_PROPERTY

METHOD metConfig
VAR_INPUT
END_VAR
fbConfigFile();

fbxSimulation 					(_usiParaNr := 1, itfConfigFb := fbConfigFile);
fbxSimulationLock				(_usiParaNr := 2, itfConfigFb := fbConfigFile);
fbrMin							(_usiParaNr := 3, itfConfigFb := fbConfigFile);
fbrMax							(_usiParaNr := 4, itfConfigFb := fbConfigFile);
fbrMinPhysical					(_usiParaNr := 5, itfConfigFb := fbConfigFile);
fbrPhysicalAlarm				(_usiParaNr := 6, itfConfigFb := fbConfigFile);
fbrSimulationValue				(_usiParaNr := 7, itfConfigFb := fbConfigFile);
fbrCorrectionValue				(_usiParaNr := 8, itfConfigFb := fbConfigFile);
fbstPhysicalUnit				(_usiParaNr := 9, itfConfigFb := fbConfigFile);
END_METHOD

PROPERTY proAlUnterlauf : BOOL
GET
proAlUnterlauf := xAlUnterlauf;
END_GET
END_PROPERTY

END_FUNCTION_BLOCK

// 21 Interface/IO_FB/AI/ITF_AI
INTERFACE ITF_AI EXTENDS ITF_IO

PROPERTY P_scfbAI_fbrPhysicalAlarm : CtaSysConfig.ITF_DATATYPE
GET
END_GET
END_PROPERTY

PROPERTY P_scfbAI_fbrSimulationValue : CtaSysConfig.ITF_DATATYPE
GET
END_GET
END_PROPERTY

PROPERTY P_scfbAI_fbstPhysicalUnit : CtaSysConfig.ITF_DATATYPE
GET
END_GET
END_PROPERTY

PROPERTY P_scfbAI_fbrCorrectionValue : CtaSysConfig.ITF_DATATYPE
GET
END_GET
END_PROPERTY

PROPERTY P_scfbAI_fbrMax : CtaSysConfig.ITF_DATATYPE
GET
END_GET
END_PROPERTY

PROPERTY P_scfbAI_fbrMin : CtaSysConfig.ITF_DATATYPE
GET
END_GET
END_PROPERTY

PROPERTY P_scfbAI_fbrMinPhysical : CtaSysConfig.ITF_DATATYPE
GET
END_GET
END_PROPERTY

PROPERTY P_All_Init : scAI_Para
SET
END_SET
END_PROPERTY

PROPERTY proAlUeberlauf : BOOL
GET
END_GET
END_PROPERTY

PROPERTY proValue : REAL
GET
END_GET
END_PROPERTY

PROPERTY proAlUnterlauf : BOOL
GET
END_GET
END_PROPERTY

METHOD FINAL metCyclicIoUpdate
VAR_INPUT
	_xOk				: BOOL;
	_rPhysicalValue 	: REAL;
	_xAlUeberlauf		: BOOL;
	_xAlUnterlauf		: BOOL;
END_VAR
END_METHOD

PROPERTY proPhysicalValue : REAL
GET
END_GET
END_PROPERTY

END_INTERFACE

// 30 Program Organization Units/IO_FB/FC/fcScaleIn
FUNCTION fcScaleIn : Real
VAR_INPUT
	rValueIn				:	REAL;
	rMin					:	REAL;
	rMax					:	REAL;
	rMinPysical				:	REAL;	
	rPysicalAlarm			:	REAL;	
	enType					: 	enIOType;
END_VAR
VAR_OUTPUT
	xAlUnterlauf	: BOOL;
END_VAR
VAR
	rPyhsicalMin		: REAL;
	rPyhsicalMax		: REAL;
END_VAR

// Prüfen des Modultyps zur definition von Min / Max
IF enType = enIOType.DC_0_10V_IN THEN	
	rPyhsicalMin		:= 0;
	rPyhsicalMax		:= 10;	
ELSIF enType = enIOType.DC_4_20mA_IN THEN
	rPyhsicalMin		:= 4;
	rPyhsicalMax		:= 20;	
ELSIF enType = enIOType.DC_0_20mA_IN THEN
	rPyhsicalMin		:= 0;
	rPyhsicalMax		:= 20;				
END_IF

// Prüfen ob die Skalierung machbar ist
IF rMax - rMin <> 0 THEN	
    // Skalieren des Messwertes
   	fcScaleIn    		:=  LIMIT(rMin,CtaAppBasic.fcScale(MAX(rValueIn,MAX(rMinPysical,rPyhsicalMin)),MAX(rMinPysical,rPyhsicalMin),rPyhsicalMax,rMin,rMax),rMax);
ELSE
	// Ausgabe des minimalen Wertes falls Skallierung nicht möglich
    fcScaleIn    		:=  MAX(rMinPysical,rPyhsicalMin);	
END_IF;
// Prüfe Physical Alarm
xAlUnterlauf  := rValueIn < rPysicalAlarm;

END_FUNCTION

// 30 Program Organization Units/IO_FB/AO/FB_AO
{attribute 'enable_dynamic_creation'}
FUNCTION_BLOCK FB_AO EXTENDS FB_IO IMPLEMENTS ITF_AO
VAR_INPUT
END_VAR
VAR_OUTPUT
END_VAR
VAR
	// Übergabewert des PGMs
	rValueIn			: 	REAL;
		
	// Calculated value
	rPhysicalValue		: 	REAL;	// Errechneter phyikalischer Wert
	
	(* Trendlog *)
	fbTrendLogrValue	:	CtaAppInfluxLog.FB_LOG_NODE_REAL;	
	(*Parameter*)
	fbrMin				: ctasysConfig.fbreAL;
	fbrMax				: ctasysConfig.fbreAL;
	fbrMinPhysical		: ctasysConfig.fbreAL;
	fbrSimulationValue	: ctasysConfig.fbreAL;	
END_VAR

PROPERTY proIsBOOL_IO : BOOL
GET
proIsBOOL_IO := FALSE;
END_GET
END_PROPERTY

PROPERTY P_All_Init : scAO_Para
SET
fbxSimulationLock._WertInit := P_All_Init.xSimulationLock;
fbrMin._WertInit			:= P_All_Init.rMin;
fbrMax._WertInit			:= P_All_Init.rMax;
fbrMinPhysical._WertInit	:= P_All_Init.rMinPhysical;
END_SET
END_PROPERTY

PROPERTY P_scfbAO_fbrMin : CtaSysConfig.ITF_DATATYPE
GET
P_scfbAO_fbrMin := fbrMin;
END_GET
END_PROPERTY

PROPERTY P_scfbAO_fbrMax : CtaSysConfig.ITF_DATATYPE
GET
P_scfbAO_fbrMax := fbrMax;
END_GET
END_PROPERTY

PROPERTY P_scfbAO_fbrSimulationValue : CtaSysConfig.ITF_DATATYPE
GET
P_scfbAO_fbrSimulationValue := fbrSimulationValue;
END_GET
END_PROPERTY

PROPERTY P_scfbAO_fbrMinPhysical : CtaSysConfig.ITF_DATATYPE
GET
P_scfbAO_fbrMinPhysical := fbrMinPhysical;
END_GET
END_PROPERTY

PROPERTY proValue : REAL
GET
proValue := rPhysicalValue;
END_GET
SET
rValueIn := proValue;
END_SET
END_PROPERTY

METHOD FINAL metCyclicIoUpdate
VAR_INPUT
	_xOk		: BOOL;
END_VAR
VAR_OUTPUT
	_rPhysicalValue : REAL;
END_VAR
(* Config *)
metConfig();

// Bei aktiver Simulation wird Simulationswert ausgegeben
IF fbxSimulation.xValue AND NOT fbxSimulationLock.xValue THEN
	// Skalierung und Übergabe des Simulationswertes 0 - 10 V
	IF enType = enIOType.DC_0_10V_OUT THEN
		rPhysicalValue := fcScaleOut(	rValueIn 			:= 	fbrSimulationValue.rValue,
										rMinPhysicalValue 	:= 	fbrMinPhysical.rValue,
										rMin 				:= 	0,
										rMax 				:= 	10,
										enType 				:= 	enType);
		fbrSimulationValue.metNewMinMax(0,10);  
	
	// Skalierung und Übergabe des Simulationswertes 4 - 20 mA	
	ELSIF  enType = enIOType.DC_4_20mA_OUT THEN
		rPhysicalValue := fcScaleOut(	rValueIn 			:= 	fbrSimulationValue.rValue,
										rMinPhysicalValue 	:= 	fbrMinPhysical.rValue,
										rMin 				:= 	4,
										rMax 				:= 	20,
										enType 				:= 	enType);
		fbrSimulationValue.metNewMinMax(4,20);  							
	// Skalierung und Übergabe des Simulationswertes 0 - 20 mA	
	ELSIF  enType = enIOType.DC_4_20mA_OUT THEN
		rPhysicalValue := fcScaleOut(	rValueIn 			:= 	fbrSimulationValue.rValue,
										rMinPhysicalValue 	:= 	fbrMinPhysical.rValue,
										rMin 				:= 	4,
										rMax 				:= 	20,
										enType 				:= 	enType);
		fbrSimulationValue.metNewMinMax(0,20);  								
	END_IF;
	(* ADD HAND Message *)
	ADD_HAND();
ELSE
	(* REM HAND Message *)
	REM_HAND();
	CASE enType OF
		enIOType.DC_0_10V_IN,enIOType.DC_0_10V_OUT:
			fbrSimulationValue.metNewMinMax(0,10); 
		enIOType.DC_0_20mA_OUT:
			fbrSimulationValue.metNewMinMax(0,20); 
		enIOType.DC_4_20mA_IN,enIOType.DC_4_20mA_OUT:
			fbrSimulationValue.metNewMinMax(4,20);
		enIOType.TEMPERATUR:
			fbrSimulationValue.metNewMinMax(-2000,8500);
		enIOType.OHM:
			fbrSimulationValue.metNewMinMax(1.0E-44,3.402823E+38);
	END_CASE	
	// Skalierung und Übergabe des PGM- Wertes
	rPhysicalValue := fcScaleOut(	rValueIn 			:= 	rValueIn,
									rMinPhysicalValue 	:= 	fbrMinPhysical.rValue,
									rMin 				:= 	fbrMin.rValue,
									rMax 				:= 	fbrMax.rValue,
									enType 				:= 	enType);
								
	fbrSimulationValue.metNewValueNoSave(rPhysicalValue);
END_IF

_rPhysicalValue := rPhysicalValue;
xOK 			:= _xOk;
	
(* TREND *)
metTrendLog();
END_METHOD

METHOD metTrendLog
IF NOT fbTrendLogrValue.ENABLE THEN
	fbTrendLogrValue.ENABLE := TRUE;
	fbTrendLogrValue.KEY	:= proLogName;
END_IF;
fbTrendLogrValue.SET_VALUE	:= rPhysicalValue;
END_METHOD

METHOD metConfig
VAR_INPUT
END_VAR
fbConfigFile();

fbxSimulation 					(_usiParaNr := 1, itfConfigFb := fbConfigFile);
fbxSimulationLock				(_usiParaNr := 2, itfConfigFb := fbConfigFile);
fbrMin							(_usiParaNr := 3, itfConfigFb := fbConfigFile);
fbrMax							(_usiParaNr := 4, itfConfigFb := fbConfigFile);
fbrMinPhysical					(_usiParaNr := 5, itfConfigFb := fbConfigFile);
fbrSimulationValue				(_usiParaNr := 7, itfConfigFb := fbConfigFile);
END_METHOD

PROPERTY proPhysicalValue : REAL
GET
proPhysicalValue := rPhysicalValue;
END_GET
END_PROPERTY

PROPERTY proPhysikalValueVisu : String(6)
GET
// Schreiben des physikalischen Wertes für Visualisierung
IF proPhysicalValue >= 10 THEN
	proPhysikalValueVisu := LEFT(TO_STRING(proPhysicalValue),4);
ELSE
	proPhysikalValueVisu := LEFT(TO_STRING(proPhysicalValue),3);
END_IF
END_GET
END_PROPERTY

END_FUNCTION_BLOCK

// 21 Interface/IO_FB/AO/ITF_AO
INTERFACE ITF_AO EXTENDS ITF_IO

PROPERTY proValue : REAL
GET
END_GET
SET
END_SET
END_PROPERTY

PROPERTY proPhysicalValue : REAL
GET
END_GET
END_PROPERTY

PROPERTY P_scfbAO_fbrMax : CtaSysConfig.ITF_DATATYPE
GET
END_GET
END_PROPERTY

PROPERTY P_scfbAO_fbrMin : CtaSysConfig.ITF_DATATYPE
GET
END_GET
END_PROPERTY

PROPERTY P_scfbAO_fbrMinPhysical : CtaSysConfig.ITF_DATATYPE
GET
END_GET
END_PROPERTY

PROPERTY P_scfbAO_fbrSimulationValue : CtaSysConfig.ITF_DATATYPE
GET
END_GET
END_PROPERTY

PROPERTY P_All_Init : scAO_Para
SET
END_SET
END_PROPERTY

METHOD FINAL metCyclicIoUpdate
VAR_INPUT
	_xOk		: BOOL;
END_VAR
VAR_OUTPUT
	_rPhysicalValue : REAL;
END_VAR
END_METHOD

END_INTERFACE

// 30 Program Organization Units/IO_FB/FC/fcScaleOut
FUNCTION fcScaleOut 	: REAL
VAR_INPUT
	rValueIn			: REAL;
	rMinPhysicalValue	: REAL;
	rMin				: REAL;
	rMax				: REAL;
	enType				: enIOType;
END_VAR
VAR
	rPyhsicalMin		: REAL;
	rPyhsicalMax		: REAL;
END_VAR

// Prüfen des Modultyps zur definition von Min / Max
IF enType = enIOType.DC_0_10V_OUT THEN	
	rPyhsicalMin		:= 0;
	rPyhsicalMax		:= 10;	
ELSIF enType = enIOType.DC_4_20mA_OUT THEN
	rPyhsicalMin		:= 4;
	rPyhsicalMax		:= 20;	
ELSIF enType = enIOType.DC_0_20mA_OUT THEN
	rPyhsicalMin		:= 0;
	rPyhsicalMax		:= 20;		
END_IF

// Prüfen ob die Skalierung machbar ist
IF rMax - rMin <> 0 THEN	
    // Skalieren des Messwertes
							
   	fcScaleOut    		:=  LIMIT(MAX(rMinPhysicalValue,rPyhsicalMin),CtaAppBasic.fcScale(MAX(rValueIn,rMin),rMin,rMax,MAX(rMinPhysicalValue,rPyhsicalMin),rPyhsicalMax),rPyhsicalMax);
ELSE
	// Ausgabe des minimalen Wertes falls Skallierung nicht möglich
    fcScaleOut    		:=  MAX(rMinPhysicalValue,rPyhsicalMin);	
END_IF;

END_FUNCTION

// 21 Interface/IO_FB/DI/ITF_DI
INTERFACE ITF_DI EXTENDS ITF_IO

METHOD FINAL metCyclicIoUpdate
VAR_INPUT
	_xChannelIn : BOOL;
	_xOk		: BOOL;
END_VAR
END_METHOD

PROPERTY P_scfbDI_fbxInvert : CtaSysConfig.ITF_DATATYPE
GET
END_GET
END_PROPERTY

PROPERTY P_scfbDI_fbxSimulationValue : CtaSysConfig.ITF_DATATYPE
GET
END_GET
END_PROPERTY

PROPERTY P_All_Init : scDI_Para
SET
END_SET
END_PROPERTY

PROPERTY proValue : BOOL
GET
END_GET
END_PROPERTY

END_INTERFACE

// 21 Interface/IO_MANAGER/ITF_IO_MANAGER
INTERFACE ITF_IO_MANAGER EXTENDS  __SYSTEM.IQueryinterface

PROPERTY IMAGE : STRING
GET
END_GET
SET
END_SET
END_PROPERTY

PROPERTY AY_ITF_DEVICE_VIS : ARRAY[0..6] OF ITF_IO_DEVICE;
GET
END_GET
END_PROPERTY

PROPERTY COUNT : UINT
GET
END_GET
END_PROPERTY

END_INTERFACE

// 30 Program Organization Units/IO_MANAGER/FB_IO_MANAGER
FUNCTION_BLOCK FB_IO_MANAGER IMPLEMENTS ITF_IO_MANAGER
VAR_INPUT
END_VAR
VAR_OUTPUT
END_VAR
VAR
	_IMAGE							:	STRING;
	_COUNT							:	UINT;
	_ayITF_DEVICE					:	ARRAY[0..6] OF ITF_IO_DEVICE;
	
	_BASE_DEVICE					:	ITF_IO_DEVICE;
	_TEMP_REG_DEVICE				:	ITF_IO_DEVICE;
	_NEXT_DEVICE_LAST_GET			:	ITF_IO_DEVICE;	
END_VAR

METHOD GET_DEVICE : ITF_IO_DEVICE
VAR_INPUT
	_usiDeviceNr	: 	USINT;
END_VAR
VAR
	_TEMP_GET_DEVICE	:	ITF_IO_DEVICE;
	udiSafe				:	UDINT;
	xNextDevInUse		:	BOOL;
END_VAR
IF TO_DINT(_usiDeviceNr) >= LOWER_BOUND(_ayITF_DEVICE,1) AND
   TO_DINT(_usiDeviceNr) <= UPPER_BOUND(_ayITF_DEVICE,1) THEN
   GET_DEVICE := _ayITF_DEVICE[_usiDeviceNr];
END_IF;

IF GET_DEVICE = 0 THEN
	IF __QUERYINTERFACE(_NEXT_DEVICE_LAST_GET,_TEMP_GET_DEVICE) THEN
		xNextDevInUse := TRUE;
	ELSIF __QUERYINTERFACE(_BASE_DEVICE,_TEMP_GET_DEVICE) THEN
		xNextDevInUse := FALSE;
	END_IF;
	
	IF __QUERYINTERFACE(_TEMP_GET_DEVICE,_TEMP_GET_DEVICE) THEN
		REPEAT 
			IF _TEMP_GET_DEVICE.DEV_NR = _usiDeviceNr THEN
				GET_DEVICE := _TEMP_GET_DEVICE;
			END_IF;
			_TEMP_GET_DEVICE	 	:= _TEMP_GET_DEVICE.LOW_SYBIL;
			_NEXT_DEVICE_LAST_GET	:= _TEMP_GET_DEVICE;
			IF _TEMP_GET_DEVICE = 0 AND xNextDevInUse THEN
				__QUERYINTERFACE(_BASE_DEVICE,_TEMP_GET_DEVICE);
				xNextDevInUse := FALSE;
			END_IF;
			udiSafe	:= udiSafe + 1;
		UNTIL GET_DEVICE <> 0 OR _TEMP_GET_DEVICE = 0 OR udiSafe >= 16#FFFFFFFE
		END_REPEAT
	ELSE
		GET_DEVICE := 0;
	END_IF;
END_IF;
END_METHOD

METHOD GET_IO : ITF_IO
VAR_INPUT
	_usiDeviceNr		:	USINT;
	_usiSlotNr			: 	USINT;
	_usiIoNr			: 	USINT;
END_VAR	
VAR
	
	_TEMP_GET_DEVICE	:	ITF_IO_DEVICE;
	_TEMP_GET_IO		:	ITF_IO;
	udiSafe				:	UDINT;
END_VAR
IF __QUERYINTERFACE(GET_DEVICE(_usiDeviceNr),_TEMP_GET_DEVICE) THEN
	GET_IO := _TEMP_GET_DEVICE.GET_IO(_usiSlotNr,_usiIoNr);
END_IF;
END_METHOD

PROPERTY AY_ITF_DEVICE_VIS : ARRAY[0..6] OF ITF_IO_DEVICE;
GET
AY_ITF_DEVICE_VIS := _ayITF_DEVICE;
END_GET
END_PROPERTY

PROPERTY COUNT : UINT
GET
COUNT := _COUNT;
END_GET
END_PROPERTY

METHOD ADD_DEVICE
VAR_INPUT
	ITF_DEVICE_IN	:	ITF_IO_DEVICE;
END_VAR
VAR
	ITF_TEMP		:	ITF_IO_DEVICE;
	ITF_TEMP_BIG	:	ITF_IO_DEVICE;
	ITF_TEMP_LOW	:	ITF_IO_DEVICE;
	xDone			:	BOOL;
END_VAR
(* Check if Valid Interface Input *)
IF __QUERYINTERFACE(ITF_DEVICE_IN,ITF_DEVICE_IN) THEN
	IF NOT CHECK_IF_DEVICE_EXIST(ITF_DEVICE_IN.DEV_NR) THEN
		IF TO_DINT(ITF_DEVICE_IN.DEV_NR) >= LOWER_BOUND(_ayITF_DEVICE,1) AND
		   TO_DINT(ITF_DEVICE_IN.DEV_NR) <= UPPER_BOUND(_ayITF_DEVICE,1) THEN
		   _ayITF_DEVICE[ITF_DEVICE_IN.DEV_NR] := ITF_DEVICE_IN;
		END_IF;
		(* Check if Valid Interface Base*)
		IF __QUERYINTERFACE(_BASE_DEVICE,_BASE_DEVICE) THEN
			(* Check if Valid Interface Temporary registration *)
			IF __QUERYINTERFACE(_TEMP_REG_DEVICE,ITF_TEMP) THEN
				REPEAT
					(* Get Big Sybil of registration *)
					IF __QUERYINTERFACE(ITF_TEMP.BIG_SYBIL,ITF_TEMP_BIG) THEN
						(* Check if Adress is Lower *)
						IF ITF_DEVICE_IN.DEV_NR <= ITF_TEMP.DEV_NR THEN
							(* Check if Adress is Bigger and update if yes*)
							IF ITF_DEVICE_IN.DEV_NR >= ITF_TEMP_BIG.DEV_NR THEN
								ITF_DEVICE_IN.BIG_SYBIL := ITF_TEMP.BIG_SYBIL;
								ITF_DEVICE_IN.LOW_SYBIL := ITF_TEMP;
								xDone	 := TRUE;							
							END_IF;
						(* Adress is Bigger update *)
						ELSE
							IF __QUERYINTERFACE(ITF_TEMP.LOW_SYBIL,ITF_TEMP_LOW) THEN
								IF 	ITF_DEVICE_IN.DEV_NR <= ITF_TEMP_LOW.DEV_NR THEN
									ITF_DEVICE_IN.LOW_SYBIL := ITF_TEMP.LOW_SYBIL;
									ITF_DEVICE_IN.BIG_SYBIL := ITF_TEMP;
									xDone	 := TRUE;
								END_IF;
							ELSE
								ITF_DEVICE_IN.LOW_SYBIL := ITF_TEMP.LOW_SYBIL;
								ITF_DEVICE_IN.BIG_SYBIL := ITF_TEMP;
								xDone	 := TRUE;
								(* Update Registation Job if temp is the last one *)
								IF ITF_TEMP = _TEMP_REG_DEVICE THEN
									_TEMP_REG_DEVICE := ITF_DEVICE_IN;
									_TEMP_REG_DEVICE.LOW_SYBIL := 0;
								END_IF;
							END_IF;
						END_IF;
					(* Interface is same as the Base*)
					ELSIF ITF_TEMP = _BASE_DEVICE THEN
						(* Check if the Input Interface needs to be the new base*)
						IF ITF_DEVICE_IN.DEV_NR <= ITF_TEMP.DEV_NR THEN 
							ITF_DEVICE_IN.LOW_SYBIL := ITF_TEMP;
							_BASE_DEVICE 				:= ITF_DEVICE_IN;
							_BASE_DEVICE.BIG_SYBIL 	:= 0;
							xDone	 				:= TRUE; 
						ELSE
							(* Update Registation Job if temp is the last one *)
							IF ITF_TEMP = _TEMP_REG_DEVICE THEN
								_TEMP_REG_DEVICE				:= ITF_DEVICE_IN;
								_TEMP_REG_DEVICE.LOW_SYBIL 	:= 0;
							END_IF
							ITF_DEVICE_IN.LOW_SYBIL := _BASE_DEVICE.LOW_SYBIL;
							_BASE_DEVICE.LOW_SYBIL 	:= ITF_DEVICE_IN;
						END_IF;
					END_IF;
					(* Get Next Interface to Check*)
					__QUERYINTERFACE(ITF_TEMP.BIG_SYBIL,ITF_TEMP);
				UNTIL xDone OR ITF_TEMP = 0 
				END_REPEAT
			ELSE
				(* Set Base Low sybill on second call*)
				_BASE_DEVICE.LOW_SYBIL 	:= ITF_DEVICE_IN;
				_TEMP_REG_DEVICE			:= ITF_DEVICE_IN;		
			END_IF;		
		ELSE
			(* Set Base on first call*)
			_BASE_DEVICE 		:= ITF_DEVICE_IN;
			_TEMP_REG_DEVICE 	:= ITF_DEVICE_IN;
		END_IF;
		(* Count Jobs *)
		_COUNT := _COUNT + 1;
	END_IF;
END_IF;
END_METHOD

METHOD CHECK_IF_DEVICE_EXIST : BOOL
VAR_INPUT
	_usiDeviceNr			: 	USINT;
END_VAR
VAR
	_TEMP_CHK_DEVICE	:	ITF_IO_DEVICE;
	udiSafe			:	UDINT;
END_VAR
IF __QUERYINTERFACE(_BASE_DEVICE,_TEMP_CHK_DEVICE) THEN
	REPEAT 
		IF _TEMP_CHK_DEVICE.DEV_NR = _usiDeviceNr THEN
			CHECK_IF_DEVICE_EXIST := TRUE;
		END_IF;
		_TEMP_CHK_DEVICE := _TEMP_CHK_DEVICE.LOW_SYBIL;
		udiSafe	:= udiSafe + 1;
	UNTIL CHECK_IF_DEVICE_EXIST OR _TEMP_CHK_DEVICE = 0 OR udiSafe >= 16#FFFFFFFE
	END_REPEAT
ELSE
	CHECK_IF_DEVICE_EXIST := FALSE;
END_IF
END_METHOD

PROPERTY IMAGE : STRING
GET
IMAGE := _IMAGE;
END_GET
SET
_IMAGE := IMAGE;
END_SET
END_PROPERTY

METHOD CHECK_SLOT : BOOL
VAR_INPUT
	_usiDeviceNr	: 	USINT;
	_usiSlotNr		: 	USINT;
	enCheckIoIn		:	enCheckIo;
	enSimIoTypeIn	:	enIOType := enIOType.Unknown;
	usiAnzIoType	:	USINT;
END_VAR
VAR
	ITF_DEVICE		: 	ITF_IO_DEVICE;
END_VAR
ITF_DEVICE := GET_DEVICE(_usiDeviceNr);
IF __QUERYINTERFACE(ITF_DEVICE,ITF_DEVICE) THEN
	CHECK_SLOT := ITF_DEVICE.CHECK_SLOT(_usiSlotNr,enCheckIoIn,usiAnzIoType);
	ITF_DEVICE.SIM_IO_TYPE(_usiSlotNr,enSimIoTypeIn,usiAnzIoType,'');
ELSE
	CHECK_SLOT := FALSE;
END_IF;
END_METHOD

END_FUNCTION_BLOCK

// 30 Program Organization Units/FC/FC_VIS_IO_TABLE
FUNCTION FC_VIS_IO_TABLE : ARRAY[1..18] OF ITF_IO_TABLE
VAR_INPUT
	ITF_IO_SLOT_IN	:	ITF_IO_SLOT;	
END_VAR
VAR_OUTPUT
	iMax				:	INT;
END_VAR
VAR
	ITF_TEMP_SLOT		:	ITF_IO_SLOT;
	ITF_LOW_IO_SYBIL	:	ITF_IO;
	usiCOUNT			:	USINT;
	usiFor				:	USINT;
END_VAR

iMax 		:= 0;
usiCOUNT 	:= 1;
IF __QUERYINTERFACE(ITF_IO_SLOT_IN,ITF_TEMP_SLOT) THEN
	REPEAT
		IF ITF_TEMP_SLOT.COUNT > 0 THEN
			FOR usiFor := 1 TO ITF_TEMP_SLOT.COUNT DO
				IF __QUERYINTERFACE(ITF_TEMP_SLOT.GET_IO(usiFor),FC_VIS_IO_TABLE[usiCOUNT]) THEN
					usiCOUNT := usiCOUNT + 1;
					iMax	 := iMax + 1;
					IF usiCOUNT >= 19 THEN
						EXIT;
					END_IF;
				END_IF;
			END_FOR;
		END_IF;
		ITF_TEMP_SLOT := ITF_TEMP_SLOT.LOW_SYBIL;
	UNTIL usiCOUNT >= 19 OR ITF_TEMP_SLOT = 0
	END_REPEAT
END_IF;

END_FUNCTION

// 40 Visualizations/IO_FB/AI/SimAI_Temp
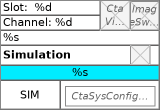
VISUALIZATION SimAI_Temp  // 160x110
VAR_INPUT
	ITF_AI : ITF_AI;
END_VAR
    RoundedRectangle (0,80 60x30)
    RoundedRectangle (60,80 100x30)
    Frame (0,0 160x45)
        shows ModulInfos(ITF_IO := ITF_AI)
    Frame (0,45 160x20)
        shows SimulationInfos(ITF_IO_IN := ITF_AI)
    Textfield (0,65 160x15), "%s", text variable: ITF_AI.proPhysikalValueVisu
    Frame (0,80 60x30), invisible if: ITF_AI.proIsSimLocked, input disabled if: ITF_AI.proIsSimLocked
        shows SimIO(ITF_IO := ITF_AI)
    Frame (65,86 90x20), invisible if: ITF_AI.proIsSimLocked, input disabled if: ITF_AI.proIsSimLocked
        shows CtaSysConfig.visREAL(visfbREALIn := ITF_AI.P_scfbAI_fbrSimulationValue)
END_VISUALIZATION

// 40 Visualizations/IO_FB/AI/SimAI
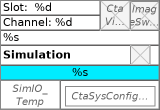
VISUALIZATION SimAI  // 160x110
VAR_INPUT	
	ITF_AI : ITF_AI;
END_VAR
    Frame (0,0 160x110), invisible if: NOT __QUERYINTERFACE(ITF_AI,ITF_AI)
        shows SimAI_Temp_Querry(ITF_AI := ITF_AI)
END_VISUALIZATION

// 40 Visualizations/IO_FB/AO/SimAO_Temp
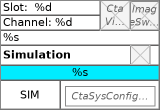
VISUALIZATION SimAO_Temp  // 160x110
VAR_INPUT
	ITF_AO : ITF_AO;
END_VAR
    RoundedRectangle (0,80 60x30)
    RoundedRectangle (60,80 100x30)
    Frame (0,0 160x45)
        shows ModulInfos(ITF_IO := ITF_AO)
    Frame (0,45 160x20)
        shows SimulationInfos(ITF_IO_IN := ITF_AO)
    Textfield (0,65 160x15), "%s", text variable: ITF_AO.proPhysikalValueVisu
    Frame (0,80 60x30), invisible if: ITF_AO.proIsSimLocked, input disabled if: ITF_AO.proIsSimLocked
        shows SimIO(ITF_IO := ITF_AO)
    Frame (65,86 90x20), invisible if: ITF_AO.proIsSimLocked, input disabled if: ITF_AO.proIsSimLocked
        shows CtaSysConfig.visREAL(visfbREALIn := ITF_AO.P_scfbAO_fbrSimulationValue)
END_VISUALIZATION

// 40 Visualizations/IO_FB/AO/SimAO
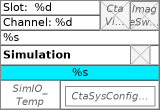
VISUALIZATION SimAO  // 160x110
VAR_INPUT	
	ITF_AO : ITF_AO;
END_VAR
    Frame (0,0 160x110), invisible if: NOT __QUERYINTERFACE(ITF_AO,ITF_AO)
        shows SimAO_Temp_Querry(ITF_AO := ITF_AO)
END_VISUALIZATION

// 40 Visualizations/IO_FB/DI/SimDI
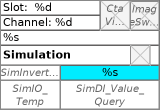
VISUALIZATION SimDI  // 160x110
VAR_INPUT	
	ITF_DI : ITF_DI;
END_VAR
    Frame (0,0 160x110), invisible if: NOT __QUERYINTERFACE(ITF_DI,ITF_DI)
        shows SimDI_Temp_Querry(ITF_DI := ITF_DI)
END_VISUALIZATION

// 40 Visualizations/IO_FB/DI/SimDI_Temp
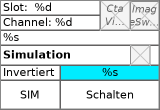
VISUALIZATION SimDI_Temp  // 160x110
VAR_INPUT
	ITF_DI : ITF_DI;
END_VAR
VAR
	ITF_BOOL : CtaSysConfig.ITF_BOOL;
END_VAR
    RoundedRectangle (0,80 60x30)
    Textfield (60,65 100x15), "%s", text variable: ITF_DI.proPhysikalValueVisu
    Frame (0,0 160x45)
        shows ModulInfos(ITF_IO := ITF_DI)
    Frame (0,45 160x20)
        shows SimulationInfos(ITF_IO_IN := ITF_DI)
    Frame (0,80 60x30), invisible if: ITF_DI.proIsSimLocked, input disabled if: ITF_DI.proIsSimLocked
        shows SimIO(ITF_IO := ITF_DI)
    Frame (0,65 60x15), invisible if: NOT __QUERYINTERFACE(ITF_DI.P_scfbDI_fbxInvert,ITF_BOOL)
        shows SimInvert(ITF_BOOL := ITF_BOOL)
    Frame (60,80 100x30), invisible if: ITF_DI.proIsSimLocked, input disabled if: ITF_DI.proIsSimLocked
        shows SimDI_Value(ITF_DI := ITF_DI)
END_VISUALIZATION

// 40 Visualizations/IO_FB/DO/SimDO_Temp
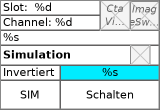
VISUALIZATION SimDO_Temp  // 160x110
VAR_INPUT	
	ITF_DO : ITF_DO;
END_VAR
VAR
	ITF_BOOL : CtaSysConfig.ITF_BOOL;
END_VAR
    RoundedRectangle (0,80 60x30)
    Frame (0,0 160x45)
        shows ModulInfos(ITF_IO := ITF_DO)
    Frame (0,45 160x20)
        shows SimulationInfos(ITF_IO_IN := ITF_DO)
    Textfield (60,65 100x15), "%s", text variable: ITF_DO.proPhysikalValueVisu
    Frame (0,80 60x30), invisible if: ITF_DO.proIsSimLocked, input disabled if: ITF_DO.proIsSimLocked
        shows SimIO(ITF_IO := ITF_DO)
    Frame (60,80 100x30), invisible if: ITF_DO.proIsSimLocked, input disabled if: ITF_DO.proIsSimLocked
        shows SimDO_Value(ITF_DO := ITF_DO)
    Frame (0,65 60x15), invisible if: NOT __QUERYINTERFACE(ITF_DO.P_scfbDO_fbxInvert,ITF_BOOL)
        shows SimInvert(ITF_BOOL := ITF_BOOL)
END_VISUALIZATION

// 40 Visualizations/IO_FB/DO/SimDO
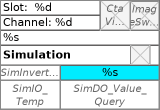
VISUALIZATION SimDO  // 160x110
VAR_INPUT	
	ITF_DO : ITF_DO;
END_VAR
    Frame (0,0 160x110), invisible if: NOT __QUERYINTERFACE(ITF_DO,ITF_DO)
        shows SimDO_Temp_Querry(ITF_DO := ITF_DO)
END_VISUALIZATION

// 40 Visualizations/IO_MANAGER/DEVICE/VIS_DEVICE
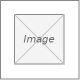
VISUALIZATION VIS_DEVICE  // 80x80
VAR_INPUT
	ITF_IO_DEVICE_IN	:	ITF_IO_DEVICE;	
END_VAR
    Frame (0,0 80x80), invisible if: NOT __QUERYINTERFACE(ITF_IO_DEVICE_IN,ITF_IO_DEVICE_IN)
        shows VIS_DEVICE_QUERY(ITF_IO_DEVICE_IN := ITF_IO_DEVICE_IN)
END_VISUALIZATION

// 40 Visualizations/IO_FB/Simulation/Simulation
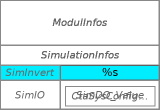
VISUALIZATION Simulation  // 160x110
VAR_INPUT	
	ITF_IO : ITF_IO;
END_VAR

VAR
	ITF_DI 	:	ITF_DI;
	ITF_DO 	:	ITF_DO;
	ITF_AI	:	ITF_AI;
	ITF_AO	:	ITF_AO;
END_VAR
    Frame (0,0 160x110), invisible if: NOT __QUERYINTERFACE(ITF_IO,ITF_DI)
        shows SimDI(ITF_DI := ITF_DI)
    Frame (0,0 160x110), invisible if: NOT __QUERYINTERFACE(ITF_IO,ITF_AI)
        shows SimAI(ITF_AI := ITF_AI)
    Frame (0,0 160x110), invisible if: NOT __QUERYINTERFACE(ITF_IO,ITF_AO)
        shows SimAO(ITF_AO := ITF_AO)
    Frame (0,0 160x110), invisible if: NOT __QUERYINTERFACE(ITF_IO,ITF_DO)
        shows SimDO(ITF_DO := ITF_DO)
END_VISUALIZATION

// 40 Visualizations/IO_FB/Simulation/ModulInfos
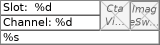
VISUALIZATION ModulInfos  // 160x45
VAR_INPUT	
	ITF_IO : ITF_IO;
END_VAR
    Textfield (0,0 100x15), "Slot: %d", text variable: ITF_IO.SLOT_NR
    Textfield (0,15 100x15), "Channel: %d", text variable: ITF_IO.IO_NR
    Textfield (0,30 160x15), "%s", text list: 'txtIOType', text index: ITF_IO.IO_TYPE
    Rectangle (130,0 30x30)
    ImageSwitcher (130,1 29x29), variable: ITF_IO.proOK, input disabled if: TRUE, background image: CtaVisSymbols.ImagePool.check_green, image: CtaVisSymbols.ImagePool.CtaError, behaviour: TOGGLE
    Rectangle (100,0 30x30)
    Image (100,0 30x30), image: CtaVisSymbols.ImagePool.gear
        OnMouseClick:  Dialog=DIA_IO_CONFIG, Parameters={ITF_IO_IN: ITF_IO}, OpenModal=True, OpenCentered=True
END_VISUALIZATION

// 40 Visualizations/IO_FB/Simulation/SimulationInfos
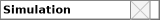
VISUALIZATION SimulationInfos  // 160x20
VAR_INPUT
	ITF_IO_IN : ITF_IO;
END_VAR
    Rectangle (0,0 160x20)
    Label (0,0 100x20), "Simulation", invisible if: ITF_IO_IN.proIsSimLocked
    Image (130,0 20x20)
        p84334746: ITF_IO_IN.proSimVisu
END_VISUALIZATION

// 40 Visualizations/IO_FB/Parameter/VIS_IO_PARAMETER_BASE
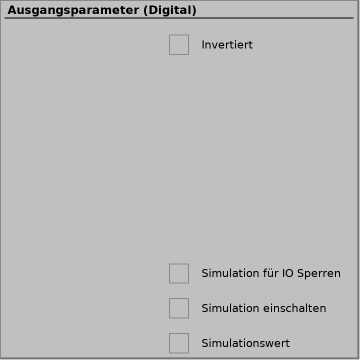
VISUALIZATION VIS_IO_PARAMETER_BASE  // 360x360
VAR_INPUT
    ITF_IO_IN 	: 	ITF_IO;
END_VAR
VAR
	ITF_AI 		:	ITF_AI;
	ITF_DI		:	ITF_DI;
	ITF_AO		:	ITF_AO;
	ITF_DO		:	ITF_DO;
END_VAR
    Frame (0,0 360x360), invisible if: NOT __QUERYINTERFACE(ITF_IO_IN,ITF_AI)
        shows VIS_PARAMETER_AI(ITF_AI_IN := ITF_AI)
        shows VIS_PARAMETER_AO(ITF_AO_IN := ITF_AO)
        shows VIS_PARAMETER_DI(ITF_DI_IN := ITF_DI)
        shows VIS_PARAMETER_DO(ITF_DO_IN := ITF_DO)
        p1531675999: ITF_SENSOR_IN.proThisReference
    Frame (0,0 360x360), invisible if: NOT __QUERYINTERFACE(ITF_IO_IN,ITF_AO)
        shows VIS_PARAMETER_AO(ITF_AO_IN := ITF_AO)
        shows VIS_PARAMETER_AO(ITF_AO_IN := ITF_AO)
        shows VIS_PARAMETER_DI(ITF_DI_IN := ITF_DI)
        shows VIS_PARAMETER_DO(ITF_DO_IN := ITF_DO)
        p1531675999: ITF_SENSOR_IN.proThisReference
    Frame (0,0 360x360), invisible if: NOT __QUERYINTERFACE(ITF_IO_IN,ITF_DI)
        shows VIS_PARAMETER_DI(ITF_DI_IN := ITF_DI)
        shows VIS_PARAMETER_AO(ITF_AO_IN := ITF_AO)
        shows VIS_PARAMETER_DI(ITF_DI_IN := ITF_DI)
        shows VIS_PARAMETER_DO(ITF_DO_IN := ITF_DO)
        p1531675999: ITF_SENSOR_IN.proThisReference
    Frame (0,0 360x360), invisible if: NOT __QUERYINTERFACE(ITF_IO_IN,ITF_DO)
        shows VIS_PARAMETER_DO(ITF_DO_IN := ITF_DO)
        shows VIS_PARAMETER_AO(ITF_AO_IN := ITF_AO)
        shows VIS_PARAMETER_DI(ITF_DI_IN := ITF_DI)
        shows VIS_PARAMETER_DO(ITF_DO_IN := ITF_DO)
        p1531675999: ITF_SENSOR_IN.proThisReference
END_VISUALIZATION

// 40 Visualizations/IO_FB/Parameter/Parameter_AI/VIS_PARAMETER_AI
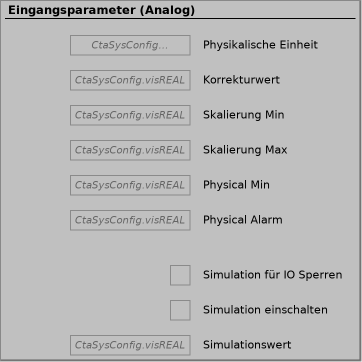
VISUALIZATION VIS_PARAMETER_AI  // 362x362
VAR_INPUT
    ITF_AI_IN	:  	ITF_AI;
END_VAR
    Frame (0,0 362x362), invisible if: NOT __QUERYINTERFACE(ITF_AI_IN,ITF_AI_IN)
        shows VIS_PARAMETER_TEMP_AI(ITF_AI_IN := ITF_AI_IN)
END_VISUALIZATION

// 40 Visualizations/IO_FB/Parameter/Parameter_AI/VIS_PARAMETER_TEMP_AI
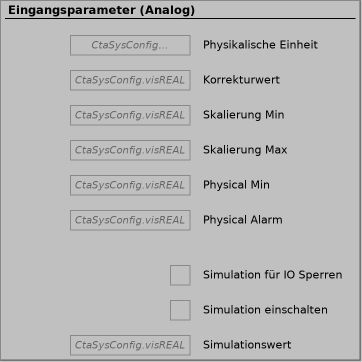
VISUALIZATION VIS_PARAMETER_TEMP_AI  // 362x362
VAR_INPUT
    ITF_AI_IN	:  	ITF_AI;
END_VAR
    RoundedRectangle (0,0 360x360)
    Label (5,0 350x20), "Eingangsparameter (Analog)"
    Line (5,18) (355,18)
    Frame (70,35 120x20), invisible if: ITF_AI_IN.IO_TYPE = 7
        shows CtaSysConfig.visSTRING40(visfbSTRING40In := ITF_AI_IN.P_scfbAI_fbstPhysicalUnit)
    Label (200,35 150x20), "Physikalische Einheit", invisible if: ITF_AI_IN.IO_TYPE = 7
    Frame (70,70 120x20)
        shows CtaSysConfig.visREAL(visfbREALIn := ITF_AI_IN.P_scfbAI_fbrCorrectionValue, stPhysikalischeEinheit := CtaSysConfig.fcGetValueFromDataType(ITF_AI_IN.P_scfbAI_fbstPhysicalUnit))
    Label (200,70 150x20), "Korrekturwert"
    Frame (70,105 120x20), invisible if: ITF_AI_IN.IO_TYPE = enIOType.TEMPERATUR OR ITF_AI_IN.IO_TYPE = enIOType.OHM
        shows CtaSysConfig.visREAL(visfbREALIn := ITF_AI_IN.P_scfbAI_fbrMin, stPhysikalischeEinheit := CtaSysConfig.fcGetValueFromDataType(ITF_AI_IN.P_scfbAI_fbstPhysicalUnit))
    Label (200,105 150x20), "Skalierung Min", invisible if: ITF_AI_IN.IO_TYPE = enIOType.TEMPERATUR OR ITF_AI_IN.IO_TYPE = enIOType.OHM
    Frame (70,140 120x20), invisible if: ITF_AI_IN.IO_TYPE = enIOType.TEMPERATUR OR ITF_AI_IN.IO_TYPE = enIOType.OHM
        shows CtaSysConfig.visREAL(visfbREALIn := ITF_AI_IN.P_scfbAI_fbrMax, stPhysikalischeEinheit := CtaSysConfig.fcGetValueFromDataType(ITF_AI_IN.P_scfbAI_fbstPhysicalUnit))
    Label (200,140 150x20), "Skalierung Max", invisible if: ITF_AI_IN.IO_TYPE = enIOType.TEMPERATUR OR ITF_AI_IN.IO_TYPE = enIOType.OHM
    Frame (70,175 120x20), invisible if: ITF_AI_IN.IO_TYPE <> 5
        shows CtaSysConfig.visREAL(visfbREALIn := ITF_AI_IN.P_scfbAI_fbrMinPhysical, stPhysikalischeEinheit := 'V')
    Label (200,175 150x20), "Physical Min", invisible if: ITF_AI_IN.IO_TYPE <> 5
    Frame (70,210 120x20), invisible if: ITF_AI_IN.IO_TYPE <> 5
        shows CtaSysConfig.visREAL(visfbREALIn := ITF_AI_IN.P_scfbAI_fbrPhysicalAlarm, stPhysikalischeEinheit := 'V')
    Label (200,210 150x20), "Physical Alarm", invisible if: ITF_AI_IN.IO_TYPE <> 5
    Frame (70,335 120x20), invisible if: CtaSysConfig.fcGetEnumerationId(ITF_AI_IN.P_scfbIO_fbxSimulationLock) = 1
        shows CtaSysConfig.visREAL(visfbREALIn := ITF_AI_IN.P_scfbAI_fbrSimulationValue)
    Label (200,335 150x20), "Simulationswert", invisible if: CtaSysConfig.fcGetEnumerationId(ITF_AI_IN.P_scfbIO_fbxSimulationLock) = 1
    Label (200,300 150x20), "Simulation einschalten", invisible if: CtaSysConfig.fcGetEnumerationId(ITF_AI_IN.P_scfbIO_fbxSimulationLock) = 1
    Label (200,265 150x20), "Simulation für IO Sperren"
    Frame (170,265 20x20)
        shows CtaSysConfig.visBOOL(visfbBOOLIn := ITF_AI_IN.P_scfbIO_fbxSimulationLock)
    Frame (170,300 20x20), invisible if: CtaSysConfig.fcGetEnumerationId(ITF_AI_IN.P_scfbIO_fbxSimulationLock) = 1
        shows CtaSysConfig.visBOOL(visfbBOOLIn := ITF_AI_IN.P_scfbIO_Simulation)
    Textfield (295,335 60x20), text list: 'txtPhysicalUnit', text index: TO_STRING(TO_INT(ITF_AI_IN.IO_TYPE))
END_VISUALIZATION

// 40 Visualizations/IO_FB/Parameter/Parameter_DI/VIS_PARAMETER_DI
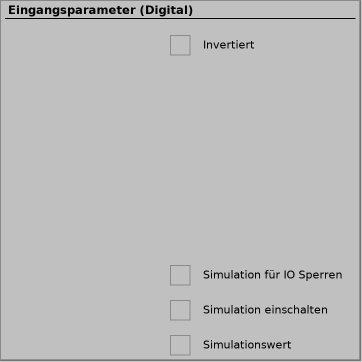
VISUALIZATION VIS_PARAMETER_DI  // 362x362
VAR_INPUT
    ITF_DI_IN	:  	ITF_DI;
END_VAR
    Frame (0,0 362x362), invisible if: NOT __QUERYINTERFACE(ITF_DI_IN,ITF_DI_IN)
        shows VIS_PARAMETER_TEMP_DI(ITF_DI_IN := ITF_DI_IN)
        pReferences[0]: IO_REF_IN=ITF_AI_IN.proThisRef_AI
END_VISUALIZATION

// 40 Visualizations/IO_FB/Parameter/Parameter_DI/VIS_PARAMETER_TEMP_DI
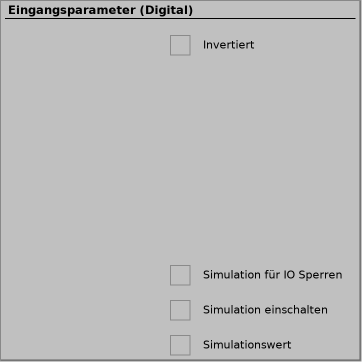
VISUALIZATION VIS_PARAMETER_TEMP_DI  // 362x362
VAR_INPUT
    ITF_DI_IN	:  	ITF_DI;
END_VAR
    RoundedRectangle (0,0 360x360)
    Label (5,0 350x20), "Eingangsparameter (Digital)"
    Line (5,18) (355,18)
    Frame (170,35 20x20)
        shows CtaSysConfig.visBOOL(visfbBOOLIn := ITF_DI_IN.P_scfbDI_fbxInvert)
    Label (200,35 150x20), "Invertiert"
    Frame (170,335 20x20), invisible if: CtaSysConfig.fcGetEnumerationId(ITF_DI_IN.P_scfbIO_fbxSimulationLock) = 1
        shows CtaSysConfig.visBOOL(visfbBOOLIn := ITF_DI_IN.P_scfbDI_fbxSimulationValue)
    Label (200,335 150x20), "Simulationswert", invisible if: CtaSysConfig.fcGetEnumerationId(ITF_DI_IN.P_scfbIO_fbxSimulationLock) = 1
    Frame (170,265 20x20)
        shows CtaSysConfig.visBOOL(visfbBOOLIn := ITF_DI_IN.P_scfbIO_fbxSimulationLock)
    Label (200,300 150x20), "Simulation einschalten", invisible if: CtaSysConfig.fcGetEnumerationId(ITF_DI_IN.P_scfbIO_fbxSimulationLock) = 1
    Label (200,265 150x20), "Simulation für IO Sperren"
    Frame (170,300 20x20), invisible if: CtaSysConfig.fcGetEnumerationId(ITF_DI_IN.P_scfbIO_fbxSimulationLock) = 1
        shows CtaSysConfig.visBOOL(visfbBOOLIn := ITF_DI_IN.P_scfbIO_Simulation)
END_VISUALIZATION

// 40 Visualizations/IO_FB/AI/SimAI_Temp_Querry
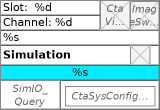
VISUALIZATION SimAI_Temp_Querry  // 160x110
VAR_INPUT
	ITF_AI : ITF_AI;
END_VAR
    Frame (0,0 160x110)
        shows SimAI_Temp(ITF_AI := ITF_AI)
END_VISUALIZATION

// 40 Visualizations/IO_FB/AO/SimAO_Temp_Querry
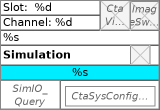
VISUALIZATION SimAO_Temp_Querry  // 160x110
VAR_INPUT
	ITF_AO : ITF_AO;
END_VAR
    Frame (0,0 160x110)
        shows SimAO_Temp(ITF_AO := ITF_AO)
END_VISUALIZATION

// 40 Visualizations/IO_FB/Parameter/Parameter_AO/VIS_PARAMETER_AO
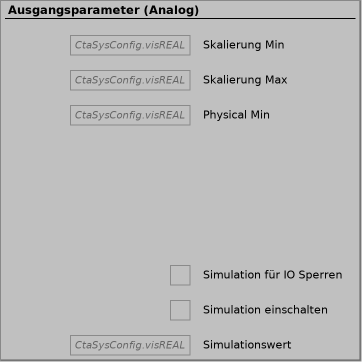
VISUALIZATION VIS_PARAMETER_AO  // 362x362
VAR_INPUT
    ITF_AO_IN	:  	ITF_AO;
END_VAR
    Frame (0,0 362x362), invisible if: NOT __QUERYINTERFACE(ITF_AO_IN,ITF_AO_IN)
        shows VIS_PARAMETER_TEMP_AO(ITF_AO_IN := ITF_AO_IN)
END_VISUALIZATION

// 40 Visualizations/IO_FB/Parameter/Parameter_AO/VIS_PARAMETER_TEMP_AO
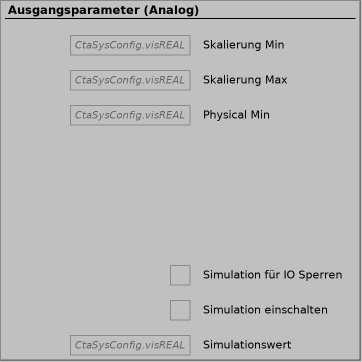
VISUALIZATION VIS_PARAMETER_TEMP_AO  // 362x362
VAR_INPUT
    ITF_AO_IN	:  	ITF_AO;
END_VAR
    RoundedRectangle (0,0 360x360)
    Label (5,0 350x20), "Ausgangsparameter (Analog)"
    Line (5,18) (355,18)
    Frame (70,35 120x20)
        shows CtaSysConfig.visREAL(visfbREALIn := ITF_AO_IN.P_scfbAO_fbrMin)
    Label (200,35 150x20), "Skalierung Min"
    Frame (70,70 120x20)
        shows CtaSysConfig.visREAL(visfbREALIn := ITF_AO_IN.P_scfbAO_fbrMax)
    Label (200,70 150x20), "Skalierung Max"
    Frame (70,105 120x20)
        shows CtaSysConfig.visREAL(visfbREALIn := ITF_AO_IN.P_scfbAO_fbrMinPhysical)
    Label (200,105 150x20), "Physical Min"
    Frame (70,335 120x20), invisible if: CtaSysConfig.fcGetEnumerationId(ITF_AO_IN.P_scfbIO_fbxSimulationLock) = 1
        shows CtaSysConfig.visREAL(visfbREALIn := ITF_AO_IN.P_scfbAO_fbrSimulationValue)
    Label (200,335 150x20), "Simulationswert", invisible if: CtaSysConfig.fcGetEnumerationId(ITF_AO_IN.P_scfbIO_fbxSimulationLock) = 1
    Frame (170,265 20x20)
        shows CtaSysConfig.visBOOL(visfbBOOLIn := ITF_AO_IN.P_scfbIO_fbxSimulationLock)
    Label (200,300 150x20), "Simulation einschalten", invisible if: CtaSysConfig.fcGetEnumerationId(ITF_AO_IN.P_scfbIO_fbxSimulationLock) = 1
    Label (200,265 150x20), "Simulation für IO Sperren"
    Frame (170,300 20x20), invisible if: CtaSysConfig.fcGetEnumerationId(ITF_AO_IN.P_scfbIO_fbxSimulationLock) = 1
        shows CtaSysConfig.visBOOL(visfbBOOLIn := ITF_AO_IN.P_scfbIO_Simulation)
    Textfield (295,335 60x20), text list: 'txtPhysicalUnit', text index: TO_STRING(TO_INT(ITF_AO_IN.IO_TYPE))
END_VISUALIZATION

// 40 Visualizations/IO_FB/Parameter/Parameter_DO/VIS_PARAMETER_DO
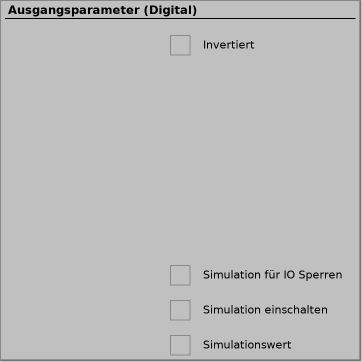
VISUALIZATION VIS_PARAMETER_DO  // 362x362
VAR_INPUT
    ITF_DO_IN	:  	ITF_DO;
END_VAR
    Frame (0,0 362x362), invisible if: NOT __QUERYINTERFACE(ITF_DO_IN,ITF_DO_IN)
        shows VIS_PARAMETER_TEMP_DO(ITF_DO_IN := ITF_DO_IN)
END_VISUALIZATION

